											IF arrAxisCtrl[AxiseNo.AxisName.TailCurlRetracting].Cmd.arrbRealPoint[1] THEN
												arrAxisCtrl[AxiseNo.AxisName.TailCurlRetracting].Cmd.iGoSetPos:=0;
												//TailCurlRetMark:=FALSE;//尾卷夹电芯伸缩力矩判断标志
											ELSE
												arrAxisCtrl[AxiseNo.AxisName.TailCurlRetracting].Cmd.iGoSetPos:=1;//尾卷夹电芯伸缩移至初始位
												//TailCurlRetMark:=TRUE;//尾卷夹电芯伸缩力矩判断标志
											END_IF
										END_IF				
										IF 	arrAxisCtrl[AxiseNo.AxisName.TailCurlLine].Status.Homed AND arrAxisCtrl[AxiseNo.AxisName.TailCurlLine].Status.NoMoving THEN
											IF arrAxisCtrl[AxiseNo.AxisName.TailCurlLine].Cmd.arrbRealPoint[3] THEN
												TailCurlTorMark:=FALSE;//尾卷夹电芯平移力矩判断标志位
												bFlgGMEndIng:=FALSE;//拉膜中
												arrAxisCtrl[AxiseNo.AxisName.TailCurlLine].Cmd.iGoSetPos:=0;
											ELSE
												arrAxisCtrl[AxiseNo.AxisName.TailCurlLine].Cmd.iGoSetPos:=3;//尾卷夹电芯平移至拉膜位
												bFlgGMEndIng:=TRUE;//拉膜中
												TailCurlTorMark:=TRUE;//尾卷夹电芯平移力矩判断标志位
											END_IF
										END_IF	
										
				(*					
							//验证：夹膜位更改			
										
										IF 	arrAxis[AxiseNo.AxisName.TailCurlSEPTALine].Status.Homed AND arrAxis[AxiseNo.AxisName.TailCurlSEPTALine].Status.NotMoving THEN
											IF arrAxisCtrl[AxiseNo.AxisName.TailCurlSEPTALine].Cmd.arrbRealPoint[4] THEN
												arrAxisCtrl[AxiseNo.AxisName.TailCurlSEPTALine].Cmd.iGoSetPos:=0;
												TailCurlSEPTATorMark:=FALSE;//夹膜平移力矩判断标志
											ELSE
												arrAxisCtrl[AxiseNo.AxisName.TailCurlSEPTALine].Cmd.iGoSetPos:=4;//尾卷夹膜平移至夹膜
												
												TailCurlSEPTATorMark:=TRUE;//夹膜平移力矩判断标志
											END_IF
										END_IF		
		*)
									
										
										
										IF arrAxisCtrl[AxiseNo.AxisName.TailCurlLine].Status.fSetPos<=  arrAxisPar[AxiseNo.AxisName.TailCurlLine].arrTargetPoint[8] THEN
													IF arrAxis[AxiseNo.AxisName.TailCurlWhirling].Status.Homed AND arrAxisCtrl[AxiseNo.AxisName.TailCurlWhirling].Status.NoMoving THEN
																IF arrAxisCtrl[AxiseNo.AxisName.TailCurlWhirling].Cmd.arrbRealPoint[3] THEN
																	arrAxisCtrl[AxiseNo.AxisName.TailCurlWhirling].Cmd.iGoSetPos:=0;
																ELSE
																	arrAxisCtrl[AxiseNo.AxisName.TailCurlWhirling].Cmd.iGoSetPos:=3;
																END_IF						
												END_IF											
										END_IF
										
								END_IF																	
								IF 	(* arrAxisCtrl[AxiseNo.AxisName.TailCurlSEPTALine].Cmd.arrbRealPoint[4] AND*) arrAxisCtrl[AxiseNo.AxisName.TailCurlRetracting].Cmd.arrbRealPoint[1] AND arrAxisCtrl[AxiseNo.AxisName.TailCurlLine].Cmd.arrbRealPoint[3] AND arrAxisCtrl[AxiseNo.AxisName.TailCurlWhirling].Cmd.arrbRealPoint[3] THEN
											tailCult_GearInMultiMaster.Enable:=FALSE;//启动尾卷拉膜凸轮耦合
											IF Mach_Control.WJ_b.SinStepMode THEN//尾卷单步模式
												TailCurlSinStep:=TRUE;
											ELSE
												TailCurlSinStep:=FALSE;
											END_IF
											fbGearInGMvirbEnable:=FALSE;
											arrAxisCtrl[AxiseNo.AxisName.TailCurlLine].Cmd.fOverride:=100;									
											TailCurlStep3:=160;
											LMcount:=LMcount+1;
								END_IF	
						END_IF
		
				151:	
								
								IF NOT TailCurlSinStep THEN			
										IF arrAxis[AxiseNo.AxisName.TailCurlWhirling].Status.Homed AND arrAxisCtrl[AxiseNo.AxisName.TailCurlWhirling].Status.NoMoving THEN
													IF arrAxisCtrl[AxiseNo.AxisName.TailCurlWhirling].Cmd.arrbRealPoint[3] THEN
														arrAxisCtrl[AxiseNo.AxisName.TailCurlWhirling].Cmd.iGoSetPos:=0;
														IF Mach_Control.WJ_b.SinStepMode THEN//尾卷单步模式
															TailCurlSinStep:=TRUE;
														ELSE
															TailCurlSinStep:=FALSE;
														END_IF	
														TailCurlStep3:=160;
													ELSE
														arrAxisCtrl[AxiseNo.AxisName.TailCurlWhirling].Cmd.iGoSetPos:=3;
													END_IF						
									END_IF
								END_IF
				160://左、右压刀开合至张开位
					IF NOT TailCurlSinStep THEN		
								arrAxisCtrl[AxiseNo.AxisName.TailCurlLine].Cmd.fOverride:=100;
								//Par.stDT_date.iTargetTorqueBLXS:=3;		
								IF 	arrAxisCtrl[AxiseNo.AxisName.LeftYDUpDown].Status.Homed AND arrAxisCtrl[AxiseNo.AxisName.LeftYDUpDown].Status.NoMoving THEN
									IF arrAxisCtrl[AxiseNo.AxisName.LeftYDUpDown].Cmd.arrbRealPoint[2] THEN
										arrAxisCtrl[AxiseNo.AxisName.LeftYDUpDown].Cmd.iGoSetPos:=0;
									ELSE
										arrAxisCtrl[AxiseNo.AxisName.LeftYDUpDown].Cmd.iGoSetPos:=2;//左压刀升降轴上升至下料高度
									END_IF
								END_IF					
								IF 	arrAxisCtrl[AxiseNo.AxisName.RightYDUpDown].Status.Homed AND arrAxisCtrl[AxiseNo.AxisName.RightYDUpDown].Status.NoMoving THEN
									IF arrAxisCtrl[AxiseNo.AxisName.RightYDUpDown].Cmd.arrbRealPoint[2] THEN
										arrAxisCtrl[AxiseNo.AxisName.RightYDUpDown].Cmd.iGoSetPos:=0;
									ELSE
										arrAxisCtrl[AxiseNo.AxisName.RightYDUpDown].Cmd.iGoSetPos:=2;//右压好升降上升至下料高度
									END_IF
								END_IF		
								
								IF 	arrAxisCtrl[AxiseNo.AxisName.TailCurlSEPTAUpDown].Status.Homed AND arrAxisCtrl[AxiseNo.AxisName.TailCurlSEPTAUpDown].Status.NoMoving THEN
									IF arrAxisCtrl[AxiseNo.AxisName.TailCurlSEPTAUpDown].Cmd.arrbRealPoint[2] THEN
										arrAxisCtrl[AxiseNo.AxisName.TailCurlSEPTAUpDown].Cmd.iGoSetPos:=0;
									ELSE
										arrAxisCtrl[AxiseNo.AxisName.TailCurlSEPTAUpDown].Cmd.iGoSetPos:=2;//
									END_IF
								END_IF					
								IF 	arrAxisCtrl[AxiseNo.AxisName.TailCurlUpDown].Status.Homed AND arrAxisCtrl[AxiseNo.AxisName.TailCurlUpDown].Status.NoMoving THEN
									IF arrAxisCtrl[AxiseNo.AxisName.TailCurlUpDown].Cmd.arrbRealPoint[2] THEN
										arrAxisCtrl[AxiseNo.AxisName.TailCurlUpDown].Cmd.iGoSetPos:=0;
									ELSE
										arrAxisCtrl[AxiseNo.AxisName.TailCurlUpDown].Cmd.iGoSetPos:=2;//
									END_IF
								END_IF			
								
								
								IF arrAxisCtrl[AxiseNo.AxisName.TailCurlSEPTAUpDown].Cmd.arrbRealPoint[2]  AND arrAxisCtrl[AxiseNo.AxisName.TailCurlUpDown].Cmd.arrbRealPoint[2] AND
									arrAxisCtrl[AxiseNo.AxisName.LeftYDUpDown].Cmd.arrbRealPoint[2] AND arrAxisCtrl[AxiseNo.AxisName.RightYDUpDown].Cmd.arrbRealPoint[2]  THEN
									IF Mach_Control.WJ_b.SinStepMode THEN//尾卷单步模式
										TailCurlSinStep:=TRUE;
									ELSE
										TailCurlSinStep:=FALSE;
									END_IF		
									TailCurlStep3:=170;
								END_IF
						END_IF		
	
				170:
						IF NOT TailCurlSinStep THEN	
							arrCyCtrl[arrCyNo.ElectValveName.PoleSplintVacuum_D].Cmd.bON:=TRUE;//夹膜下夹板真空	
							arrCyCtrl[arrCyNo.CylinderName.PoleSplintCy_D].Cmd.bON:=TRUE;//夹膜下夹板上升
								IF arrCyCtrl[arrCyNo.CylinderName.PoleSplintCy_D].Status.ONState THEN
									IF Mach_Control.WJ_b.SinStepMode THEN//尾卷单步模式
										TailCurlSinStep:=TRUE;
									ELSE
										TailCurlSinStep:=FALSE;
									END_IF									
									TailCurlStep3:=180;	
								END_IF	
						END_IF		
							
			180:
					
						IF NOT TailCurlSinStep THEN	
							arrCyCtrl[arrCyNo.CylinderName.PreDiaph].Cmd.bON:=TRUE;//叠台压隔膜气缸
							IF arrCyCtrl[arrCyNo.CylinderName.PreDiaph].Status.ONState THEN
										IF Mach_Control.WJ_b.SinStepMode THEN//尾卷单步模式
											TailCurlSinStep:=TRUE;
										ELSE
											TailCurlSinStep:=FALSE;
										END_IF							
										TailCurlStep3:=181;	
							END_IF	
						END_IF	
			181:						
						IF NOT TailCurlSinStep THEN	
									IF 	arrAxisCtrl[AxiseNo.AxisName.DTUpDown].Status.Homed AND arrAxisCtrl[AxiseNo.AxisName.DTUpDown].Status.NoMoving THEN
										IF arrAxisCtrl[AxiseNo.AxisName.DTUpDown].Cmd.arrbRealPoint[1] THEN
											arrAxisCtrl[AxiseNo.AxisName.DTUpDown].Cmd.iGoSetPos:=0;
												IF Mach_Control.DT_b.DT_Chesoe THEN
													DT_Readydown:=TRUE;	
												ELSE
													DT_Readydown:=FALSE;	
												END_IF
	
												IF Mach_Control.WJ_b.SinStepMode THEN//尾卷单步模式
													TailCurlSinStep:=TRUE;
												ELSE
													TailCurlSinStep:=FALSE;
												END_IF													
																								
												TailCurlStep3:=182;	
										ELSE
											arrAxisCtrl[AxiseNo.AxisName.DTUpDown].Cmd.iGoSetPos:=1;//叠台升降上升至初始位
									END_IF
							END_IF
					END_IF
			182:
						IF NOT DT_Readydown THEN
							TailCurlStep3:=185;
						END_IF
			185://左、右压刀开合移至初始位，叠台上升至初始位
						IF NOT TailCurlSinStep THEN		
									IF 	arrAxisCtrl[AxiseNo.AxisName.LeftYDLine].Status.Homed AND arrAxisCtrl[AxiseNo.AxisName.LeftYDLine].Status.NoMoving THEN
										IF arrAxisCtrl[AxiseNo.AxisName.LeftYDLine].Cmd.arrbRealPoint[1] THEN
											arrAxisCtrl[AxiseNo.AxisName.LeftYDLine].Cmd.iGoSetPos:=0;
										ELSE
											arrAxisCtrl[AxiseNo.AxisName.LeftYDLine].Cmd.iGoSetPos:=1;//左压刀开合至初始位
										END_IF
									END_IF					
									IF 	arrAxisCtrl[AxiseNo.AxisName.RightYDLine].Status.Homed AND arrAxisCtrl[AxiseNo.AxisName.RightYDLine].Status.NoMoving THEN
										IF arrAxisCtrl[AxiseNo.AxisName.RightYDLine].Cmd.arrbRealPoint[1] THEN
											arrAxisCtrl[AxiseNo.AxisName.RightYDLine].Cmd.iGoSetPos:=0;
										ELSE
											arrAxisCtrl[AxiseNo.AxisName.RightYDLine].Cmd.iGoSetPos:=1;//右压刀开合至初始位
										END_IF
									END_IF
									IF 	arrAxisCtrl[AxiseNo.AxisName.DTUpDown].Status.Homed AND arrAxisCtrl[AxiseNo.AxisName.DTUpDown].Status.NoMoving THEN
										IF arrAxisCtrl[AxiseNo.AxisName.DTUpDown].Cmd.arrbRealPoint[1] THEN
											arrAxisCtrl[AxiseNo.AxisName.DTUpDown].Cmd.iGoSetPos:=0;
										ELSE
											arrAxisCtrl[AxiseNo.AxisName.DTUpDown].Cmd.iGoSetPos:=1;//叠台升降上升至初始位
										END_IF
									END_IF
									IF 	arrAxisCtrl[AxiseNo.AxisName.LeftYDLine].Cmd.arrbRealPoint[1] AND arrAxisCtrl[AxiseNo.AxisName.RightYDLine].Cmd.arrbRealPoint[1] AND 
										arrAxisCtrl[AxiseNo.AxisName.DTUpDown].Cmd.arrbRealPoint[1] THEN
												TailCurlStep3:=190;
												IF Mach_Control.WJ_b.SinStepMode THEN//尾卷单步模式
													TailCurlSinStep:=TRUE;
												ELSE
													TailCurlSinStep:=FALSE;
												END_IF	
									END_IF	
						END_IF
				
					



				190://左、右压刀升降下降至初始位，压隔膜
						IF NOT TailCurlSinStep THEN			
									IF 	arrAxisCtrl[AxiseNo.AxisName.LeftYDUpDown].Status.Homed AND arrAxisCtrl[AxiseNo.AxisName.LeftYDUpDown].Status.NoMoving THEN
										IF arrAxisCtrl[AxiseNo.AxisName.LeftYDUpDown].Cmd.arrbRealPoint[1] THEN
											arrAxisCtrl[AxiseNo.AxisName.LeftYDUpDown].Cmd.iGoSetPos:=0;
										ELSE
											arrAxisCtrl[AxiseNo.AxisName.LeftYDUpDown].Cmd.iGoSetPos:=1;//左压刀升降轴下降至初始高度
										END_IF
									END_IF					
									IF 	arrAxisCtrl[AxiseNo.AxisName.RightYDUpDown].Status.Homed AND arrAxisCtrl[AxiseNo.AxisName.RightYDUpDown].Status.NoMoving THEN
										IF arrAxisCtrl[AxiseNo.AxisName.RightYDUpDown].Cmd.arrbRealPoint[1] THEN
											arrAxisCtrl[AxiseNo.AxisName.RightYDUpDown].Cmd.iGoSetPos:=0;
										ELSE
											arrAxisCtrl[AxiseNo.AxisName.RightYDUpDown].Cmd.iGoSetPos:=1;//右压好升降下降至初始高度
										END_IF
									END_IF				
									IF arrAxisCtrl[AxiseNo.AxisName.LeftYDUpDown].Cmd.arrbRealPoint[1] AND arrAxisCtrl[AxiseNo.AxisName.RightYDUpDown].Cmd.arrbRealPoint[1] THEN
										IF Mach_Control.WJ_b.SinStepMode THEN//尾卷单步模式
											TailCurlSinStep:=TRUE;
										ELSE
											TailCurlSinStep:=FALSE;
										END_IF											
										TailCurlStep3:=200;
										hot_time_ton.IN:=FALSE;
									END_IF
						END_IF
						
					(*200:
						Mach_Control.WJ_b.HotCut:=TRUE;//启动热切
						WJ_TON[1].IN:=TRUE;
						TailCurlStep3:=201;		
					
						
				201://热切丝加热、热切升降气缸下降，切隔膜///////////////////////////////
					IF NOT TailCurlSinStep THEN	
					arrCyCtrl[arrCyNo.CylinderName.PoleHotCutterCy].Cmd.bON:=TRUE;//隔膜热切升降气缸伸出
								IF arrCyCtrl[arrCyNo.CylinderName.PoleHotCutterCy].Status.ONState  THEN
										Mach_Control.WJ_b.HotCut:=FALSE;//启动热切
						                WJ_TON[1].IN:=FALSE;
							IF Mach_Control.WJ_b.SinStepMode THEN//尾卷单步模式
								TailCurlSinStep:=TRUE;
							ELSE
								TailCurlSinStep:=FALSE;
							END_IF							
									TailCurlStep3:=205;	
								END_IF	
					END_IF	*)
				
				
			
					
				
				
				
				
				
				205://热切升降气缸下降/////////////////////////////////////////
					IF NOT TailCurlSinStep THEN	
						arrCyCtrl[arrCyNo.CylinderName.PoleHotCutterCy].Cmd.bOFF:=TRUE;//隔膜热切升降气缸缩回	
							IF arrCyCtrl[arrCyNo.CylinderName.PoleHotCutterCy].Status.OFFState THEN
								IF Mach_Control.WJ_b.SinStepMode THEN//尾卷单步模式
									TailCurlSinStep:=TRUE;
								ELSE
									TailCurlSinStep:=FALSE;
								END_IF									
								TailCurlStep3:=206;	
							END_IF	
					END_IF		
				206://叠台真空打开
					arrCyCtrl[arrCyNo.ElectValveName.DTVacuum].Cmd.bON:=TRUE;
					arrCyCtrl[arrCyNo.ElectValveName.DTVacuum].Cmd.bOFF:=FALSE;
					TailCurlStep3:=207;	
				207:
					CellMemory[Mach_Control.WJ_b.WJ_Memory]:=CellMemory[Mach_Control.DT_b.DT_Memory];
					MEMSET(ADR(CellMemory[Mach_Control.DT_b.DT_Memory]),0,SIZEOF(CellMemory[Mach_Control.DT_b.DT_Memory]));
					TailCurlStep3:=210;
		
				210:
					
						IF NOT TailCurlSinStep THEN	
							arrCyCtrl[arrCyNo.CylinderName.PreDiaph].Cmd.bOFF:=TRUE;//
							IF arrCyCtrl[arrCyNo.CylinderName.PreDiaph].Status.OFFState THEN
								IF Mach_Control.WJ_b.SinStepMode THEN//尾卷单步模式
									TailCurlSinStep:=TRUE;
								ELSE
									TailCurlSinStep:=FALSE;
								END_IF									
								TailCurlStep3:=211;	
							END_IF	
						END_IF	
				211:
					IF 	arrAxisCtrl[AxiseNo.AxisName.TailCurlUpDown].Status.Homed AND arrAxisCtrl[AxiseNo.AxisName.TailCurlUpDown].Status.NoMoving THEN
						IF arrAxisCtrl[AxiseNo.AxisName.TailCurlUpDown].Cmd.arrbRealPoint[5] THEN
							arrAxisCtrl[AxiseNo.AxisName.TailCurlUpDown].Cmd.iGoSetPos:=0;
							TailCurlStep3:=213;	
						ELSE
							arrAxisCtrl[AxiseNo.AxisName.TailCurlUpDown].Cmd.iGoSetPos:=5;//尾卷夹膜升降轴尾卷高度
						END_IF
					END_IF		
				

				213:
						IF NOT TailCurlSinStep THEN				
						IF 	arrAxisCtrl[AxiseNo.AxisName.TailCurlLine].Status.Homed AND arrAxisCtrl[AxiseNo.AxisName.TailCurlLine].Status.NoMoving THEN
							IF arrAxisCtrl[AxiseNo.AxisName.TailCurlLine].Cmd.arrbRealPoint[7] THEN
								arrAxisCtrl[AxiseNo.AxisName.TailCurlLine].Cmd.iGoSetPos:=0;
								IF Mach_Control.WJ_b.SinStepMode THEN//尾卷单步模式
									TailCurlSinStep:=TRUE;
								ELSE
									TailCurlSinStep:=FALSE;
								END_IF									
								TailCurlStep3:=215;
							ELSE
								arrAxisCtrl[AxiseNo.AxisName.TailCurlLine].Cmd.iGoSetPos:=7;//尾卷夹电芯平移至回拉膜位
							END_IF
						END_IF	
						END_IF
  
			
						
						
                215://尾卷夹电芯平移至上尾卷电芯位，同时开始耦合
						IF NOT TailCurlSinStep THEN			
								tailCurlGearInEnable:=TRUE;//电子齿轮耦合
								IF 	tailCurl_GearIn.InGear AND arrAxisCtrl[AxiseNo.AxisName.TailCurlLine].Status.Homed AND arrAxisCtrl[AxiseNo.AxisName.TailCurlLine].Status.NoMoving AND
                                        arrAxisCtrl[AxiseNo.AxisName.LCurlingneedleLine].Cmd.arrbRealPoint[1]  AND arrAxisCtrl[AxiseNo.AxisName.SCurlingneedleLine].Cmd.arrbRealPoint[1] AND
                                       arrAxisCtrl[AxiseNo.AxisName.TailCurlWhirling].Cmd.arrbRealPoint[1]   THEN
									IF arrAxisCtrl[AxiseNo.AxisName.TailCurlLine].Cmd.arrbRealPoint[4] THEN
										arrAxisCtrl[AxiseNo.AxisName.TailCurlLine].Cmd.iGoSetPos:=0;
										tailCurlGearInEnable:=FALSE;//电子齿轮耦合
										IF Mach_Control.WJ_b.SinStepMode THEN//尾卷单步模式
											TailCurlSinStep:=TRUE;
										ELSE
											TailCurlSinStep:=FALSE;
										END_IF												
										TailCurlStep3:=217;
										TailCurlStep6:=10;//启动判断夹膜平移是否已经在安全位置叠台下料完成	
										WJ_TON[6].IN:=FALSE;
									ELSE
										arrAxisCtrl[AxiseNo.AxisName.TailCurlLine].Cmd.iGoSetPos:=4;//尾卷夹电芯平移至上尾卷电芯位
									END_IF
								END_IF		
						END_IF	
               
				217:	
					 WJ_TON[6].IN:=TRUE;
					Mach_Control.WJ_b.TailCurlSEPTALineSavePos[1]:=arrAxis[AxiseNo.AxisName.TailCurlSEPTALine].NcToPlc.ActPos;
					arrAxisCtrl[AxiseNo.AxisName.TailCurlSEPTALine].Cmd.bMoveRel:=FALSE;
					IF WJ_TON[6].Q THEN
						TailCurlStep3:=218;
						 WJ_TON[6].IN:=FALSE;
					 END_IF	
				 
				218:
				IF NOT TailCurlSinStep THEN	
				IF Mach_Control.WJ_b.TailCurlSEPTALineSavePos[1] -arrAxis[AxiseNo.AxisName.TailCurlSEPTALine].NcToPlc.ActPos>=4.9 
					AND arrAxisCtrl[AxiseNo.AxisName.TailCurlSEPTALine].Status.NoMoving THEN
						IF Mach_Control.WJ_b.SinStepMode THEN//尾卷单步模式
								TailCurlSinStep:=TRUE;
						ELSE
								TailCurlSinStep:=FALSE;
						END_IF
					TailCurlStep3:=220;
				ELSIF NOT (Mach_Control.WJ_b.TailCurlSEPTALineSavePos[1] -arrAxis[AxiseNo.AxisName.TailCurlSEPTALine].NcToPlc.ActPos >=4.9 )
						AND arrAxisCtrl[AxiseNo.AxisName.TailCurlSEPTALine].Status.NoMoving THEN
						IF NOT arrAxisCtrl[AxiseNo.AxisName.TailCurlSEPTALine].Status.Error 
							AND arrAxis[AxiseNo.AxisName.TailCurlSEPTALine].Status.Homed 
							AND arrAxisCtrl[AxiseNo.AxisName.TailCurlSEPTALine].Status.Enabled 
							AND arrAxisCtrl[AxiseNo.AxisName.TailCurlSEPTALine].Status.NoMoving THEN
								arrAxisPar[AxiseNo.AxisName.TailCurlSEPTALine].fVelocity_of_Rel:=20;
								arrAxisCtrl[AxiseNo.AxisName.TailCurlSEPTALine].Cmd.fPosition_of_Rel:=-5;
								arrAxisCtrl[AxiseNo.AxisName.TailCurlSEPTALine].Cmd.bMoveRel:=TRUE;
						END_IF
				END_IF
				END_IF
						
						
						
				220://长、短卷针旋转到初始位，长、短卷针气缸张开/////////
						IF NOT TailCurlSinStep THEN		
								arrCyCtrl[arrCyNo.ElectValveName.WJ_blow		].Cmd.bON:=	TRUE	;//	夹膜电芯吹气	
						
								arrCyCtrl[arrCyNo.CylinderName.CurlingSplintCy_L].Cmd.bOFF:=TRUE;//尾卷长卷针张开
								arrCyCtrl[arrCyNo.CylinderName.CurlingSplintCy_S].Cmd.bOFF:=TRUE;//尾卷短卷针张开
								arrCyCtrl[arrCyNo.ElectValveName.WJShortvacuum].Cmd.bON:=TRUE;//短卷针张开真空开
								IF 	arrAxisCtrl[AxiseNo.AxisName.LCurlingneedleWhirling].Status.Homed AND arrAxisCtrl[AxiseNo.AxisName.LCurlingneedleWhirling].Status.NoMoving THEN
									IF arrAxisCtrl[AxiseNo.AxisName.LCurlingneedleWhirling].Cmd.arrbRealPoint[1] THEN
										arrAxisCtrl[AxiseNo.AxisName.LCurlingneedleWhirling].Cmd.iGoSetPos:=0;
									ELSE
										arrAxisCtrl[AxiseNo.AxisName.LCurlingneedleWhirling].Cmd.iGoSetPos:=1;//长卷针旋转至初始位
									END_IF
								END_IF										
								IF 	arrAxisCtrl[AxiseNo.AxisName.SCurlingneedleWhirling].Status.Homed AND arrAxisCtrl[AxiseNo.AxisName.SCurlingneedleWhirling].Status.NoMoving THEN
									IF arrAxisCtrl[AxiseNo.AxisName.SCurlingneedleWhirling].Cmd.arrbRealPoint[1] THEN
										arrAxisCtrl[AxiseNo.AxisName.SCurlingneedleWhirling].Cmd.iGoSetPos:=0;
									ELSE
										arrAxisCtrl[AxiseNo.AxisName.SCurlingneedleWhirling].Cmd.iGoSetPos:=1;//短卷针旋转至初始位
									END_IF
								END_IF
								
								
								IF 	arrAxisCtrl[AxiseNo.AxisName.TailCurlUpDown].Status.Homed AND arrAxisCtrl[AxiseNo.AxisName.TailCurlUpDown].Status.NoMoving THEN
									IF arrAxisCtrl[AxiseNo.AxisName.TailCurlUpDown].Cmd.arrbRealPoint[5] THEN
										arrAxisCtrl[AxiseNo.AxisName.TailCurlUpDown].Cmd.iGoSetPos:=0;
									ELSE
										arrAxisCtrl[AxiseNo.AxisName.TailCurlUpDown].Cmd.iGoSetPos:=5;//尾卷夹膜升降轴尾卷高度
									END_IF
								END_IF	
								
								
								
								IF 	arrAxisCtrl[AxiseNo.AxisName.LCurlingneedleWhirling].Cmd.arrbRealPoint[1] AND 	arrAxisCtrl[AxiseNo.AxisName.SCurlingneedleWhirling].Cmd.arrbRealPoint[1] AND
									arrAxisCtrl[AxiseNo.AxisName.TailCurlUpDown].Cmd.arrbRealPoint[5]  AND 
                                    					arrCyCtrl[arrCyNo.CylinderName.CurlingSplintCy_L].Status.OFFState AND arrCyCtrl[arrCyNo.CylinderName.CurlingSplintCy_S].Status.OFFState THEN
										IF Mach_Control.WJ_b.SinStepMode THEN//尾卷单步模式
											TailCurlSinStep:=TRUE;
										ELSE
											TailCurlSinStep:=FALSE;
										END_IF	
									CurlingneedleLineEnable:=FALSE;//长、短卷针平移电子齿轮耦合启动																
									TailCurlStep3:=223;
								END_IF	
						END_IF	
                






			223://长卷针去夹电芯位
				IF NOT TailCurlSinStep THEN		
								
								IF 	arrAxisCtrl[AxiseNo.AxisName.LCurlingneedleLine].Status.Homed  
								AND arrAxisCtrl[AxiseNo.AxisName.LCurlingneedleWhirling].Cmd.arrbRealPoint[1]
								AND arrCyCtrl[arrCyNo.CylinderName.CurlingSplintCy_L].Status.OFFState
                                AND  arrAxisCtrl[AxiseNo.AxisName.LCurlingneedleWhirling].Io.biHomeSwitch  THEN
											IF arrAxisCtrl[AxiseNo.AxisName.LCurlingneedleLine].Cmd.arrbRealPoint[2] AND arrAxisCtrl[AxiseNo.AxisName.LCurlingneedleLine].Status.NoMoving  THEN
												arrAxisCtrl[AxiseNo.AxisName.LCurlingneedleLine].Cmd.iGoSetPos:=0;
											ELSE
												arrAxisCtrl[AxiseNo.AxisName.LCurlingneedleLine].Cmd.iGoSetPos:=2;
											END_IF
								ELSE
										Mach_Control.WJ_b.Error[9]:=TRUE;	//长卷针去夹电芯位时条件不满足报警													
								END_IF
										
								IF 	arrAxisCtrl[AxiseNo.AxisName.LCurlingneedleLine].Cmd.arrbRealPoint[2] AND arrAxisCtrl[AxiseNo.AxisName.LCurlingneedleWhirling].Cmd.arrbRealPoint[1]  THEN
										IF Mach_Control.WJ_b.SinStepMode THEN//尾卷单步模式
											TailCurlSinStep:=TRUE;
										ELSE
											TailCurlSinStep:=FALSE;
										END_IF																	
									TailCurlStep3:=225;
									TON_TailCurl[2].IN:=FALSE;
								END_IF	
						END_IF			
			225:
			
			
						IF NOT TailCurlSinStep THEN	
								 
													IF NOT TON_TailCurl[2].Q THEN					
																arrCyCtrl[arrCyNo.CylinderName.CurlingSplintCy_L].Cmd.bON:=TRUE;//尾卷长卷针夹紧	
																TON_TailCurl[2].IN:=TRUE;			
													ELSE
														TON_TailCurl[2].IN:=FALSE;
														IF Mach_Control.WJ_b.SinStepMode THEN//尾卷单步模式
															TailCurlSinStep:=TRUE;
														ELSE
															TailCurlSinStep:=FALSE;
														END_IF							
														TailCurlStep3:=227;	
												END_IF
									
						END_IF

			227://短卷针去夹电芯位
	
						
					IF NOT TailCurlSinStep THEN													
								IF 	arrAxisCtrl[AxiseNo.AxisName.SCurlingneedleLine].Status.Homed  
									AND arrAxisCtrl[AxiseNo.AxisName.SCurlingneedleWhirling].Cmd.arrbRealPoint[1] AND  arrCyCtrl[arrCyNo.CylinderName.CurlingSplintCy_S].Status.OFFState 
									AND  arrCyCtrl[arrCyNo.ElectValveName.WJShortvacuum].Io.DOStatus1
                                    AND  arrAxisCtrl[AxiseNo.AxisName.SCurlingneedleWhirling].Io.biHomeSwitch THEN
												IF arrAxisCtrl[AxiseNo.AxisName.SCurlingneedleLine].Cmd.arrbRealPoint[2] AND arrAxisCtrl[AxiseNo.AxisName.SCurlingneedleLine].Status.NoMoving  THEN
													arrAxisCtrl[AxiseNo.AxisName.SCurlingneedleLine].Cmd.iGoSetPos:=0;
												ELSE
													arrAxisCtrl[AxiseNo.AxisName.SCurlingneedleLine].Cmd.iGoSetPos:=2;
												END_IF
								ELSE
										Mach_Control.WJ_b.Error[10]:=TRUE;	//短卷针去夹电芯位时条件不满足报警										
												
								END_IF

								IF 		arrAxisCtrl[AxiseNo.AxisName.SCurlingneedleLine].Cmd.arrbRealPoint[2] AND arrAxisCtrl[AxiseNo.AxisName.SCurlingneedleWhirling].Cmd.arrbRealPoint[1] THEN
										IF Mach_Control.WJ_b.SinStepMode THEN//尾卷单步模式
											TailCurlSinStep:=TRUE;
										ELSE
											TailCurlSinStep:=FALSE;
										END_IF																	
									TailCurlStep3:=230;
									TON_TailCurl[4].IN:=FALSE;
								END_IF	
						END_IF		
						
			
						
				230://短卷针夹爪气缸夹紧
						IF NOT TailCurlSinStep THEN	
							     
													IF NOT TON_TailCurl[4].Q THEN
														arrCyCtrl[arrCyNo.ElectValveName.WJShortvacuum].Cmd.bOFF:=TRUE;//短卷针张开真空关
														arrCyCtrl[arrCyNo.CylinderName.CurlingSplintCy_S].Cmd.bON:=TRUE;//尾卷短卷针夹紧	
														
														TON_TailCurl[4].IN:=TRUE;							
													ELSE
														TON_TailCurl[4].IN:=FALSE;
														IF Mach_Control.WJ_b.SinStepMode THEN//尾卷单步模式
															TailCurlSinStep:=TRUE;
														ELSE
															TailCurlSinStep:=FALSE;
														END_IF							
														TailCurlStep3:=235;	
														TON_TailCurl[6].IN:=FALSE;
												END_IF
										
						END_IF
				               
				235:
				Mach_Control.WJ_b.TailCurlSEPTALineSavePos[2]:=arrAxis[AxiseNo.AxisName.TailCurlSEPTALine].NcToPlc.ActPos;
				TailCurlStep3:=238;

				238:
				IF NOT TailCurlSinStep THEN	
				IF arrAxis[AxiseNo.AxisName.TailCurlSEPTALine].NcToPlc.ActPos-Mach_Control.WJ_b.TailCurlSEPTALineSavePos[2] >=4.9 
					AND arrAxisCtrl[AxiseNo.AxisName.TailCurlSEPTALine].Status.NoMoving THEN
						IF Mach_Control.WJ_b.SinStepMode THEN//尾卷单步模式
								TailCurlSinStep:=TRUE;
						ELSE
								TailCurlSinStep:=FALSE;
						END_IF
					TailCurlStep3:=240;
				ELSIF NOT (arrAxis[AxiseNo.AxisName.TailCurlSEPTALine].NcToPlc.ActPos-Mach_Control.WJ_b.TailCurlSEPTALineSavePos[2] >=4.9 )
					AND arrAxisCtrl[AxiseNo.AxisName.TailCurlSEPTALine].Status.NoMoving THEN
						IF NOT arrAxisCtrl[AxiseNo.AxisName.TailCurlSEPTALine].Status.Error 
							AND arrAxis[AxiseNo.AxisName.TailCurlSEPTALine].Status.Homed 
							AND arrAxisCtrl[AxiseNo.AxisName.TailCurlSEPTALine].Status.Enabled 
							AND arrAxisCtrl[AxiseNo.AxisName.TailCurlSEPTALine].Status.NoMoving THEN
								arrAxisPar[AxiseNo.AxisName.TailCurlSEPTALine].fVelocity_of_Rel:=20;
								arrAxisCtrl[AxiseNo.AxisName.TailCurlSEPTALine].Cmd.fPosition_of_Rel:=5;
								arrAxisCtrl[AxiseNo.AxisName.TailCurlSEPTALine].Cmd.bMoveRel:=TRUE;
						END_IF
				END_IF
				END_IF
				
				240://尾卷夹电芯气缸开张
						IF NOT TailCurlSinStep THEN	
							arrCyCtrl[arrCyNo.ElectValveName.WJ_blow].Cmd.bOFF:=TRUE;//	夹膜电芯吹气关
							arrCyCtrl[arrCyNo.CylinderName.TailCurlSplintCy].Cmd.bOFF:=TRUE;//尾卷取料夹爪气缸张开
							TON_TailCurl[6].IN:=TRUE;
							IF arrCyCtrl[arrCyNo.CylinderName.TailCurlSplintCy].Status.OFFState AND TON_TailCurl[6].Q	THEN
								IF Mach_Control.WJ_b.SinStepMode THEN//尾卷单步模式
									TailCurlSinStep:=TRUE;
								ELSE
									TailCurlSinStep:=FALSE;
								END_IF						
								TailCurlStep3:=250;
								TON_TailCurl[6].IN:=FALSE;
							END_IF
						END_IF
				250://尾卷夹电芯平移至初始位，启动尾卷
						IF NOT TailCurlSinStep THEN			
									IF 	arrCyCtrl[arrCyNo.CylinderName.TailCurlSplintCy].Status.OFFState AND  arrAxisCtrl[AxiseNo.AxisName.TailCurlLine].Status.Homed AND arrAxisCtrl[AxiseNo.AxisName.TailCurlLine].Status.NoMoving THEN
											IF arrAxisCtrl[AxiseNo.AxisName.TailCurlLine].Cmd.arrbRealPoint[5] THEN
												TailCurlTorMark:=FALSE;//尾卷夹电芯平移力矩判断标志位
												//TailCurlStart:=TRUE;//启动尾卷
												arrAxisCtrl[AxiseNo.AxisName.TailCurlLine].Cmd.iGoSetPos:=0;
											ELSE
												arrAxisCtrl[AxiseNo.AxisName.TailCurlLine].Cmd.iGoSetPos:=5;//尾卷夹电芯平移至初始位
												TailCurlTorMark:=TRUE;//尾卷夹电芯平移力矩判断标志位
											END_IF
									END_IF	
									
									IF arrCyCtrl[arrCyNo.CylinderName.TailCurlSplintCy].Status.OFFState AND  	arrAxisCtrl[AxiseNo.AxisName.TailCurlRetracting].Status.Homed AND arrAxisCtrl[AxiseNo.AxisName.TailCurlRetracting].Status.NoMoving THEN
											IF arrAxisCtrl[AxiseNo.AxisName.TailCurlRetracting].Cmd.arrbRealPoint[1] THEN
												//TailCurlRetMark:=FALSE;//尾卷夹电芯伸缩力矩判断标志
												arrAxisCtrl[AxiseNo.AxisName.TailCurlRetracting].Cmd.iGoSetPos:=0;
											ELSE
												arrAxisCtrl[AxiseNo.AxisName.TailCurlRetracting].Cmd.iGoSetPos:=1;//尾卷夹电芯伸缩移至初始位
												//TailCurlRetMark:=TRUE;//尾卷夹电芯伸缩力矩判断标志
											END_IF
									END_IF		
									
									IF 		arrAxisCtrl[AxiseNo.AxisName.TailCurlLine].Cmd.arrbRealPoint[5] AND arrAxisCtrl[AxiseNo.AxisName.TailCurlLine].Status.NoMoving AND
											 arrAxisCtrl[AxiseNo.AxisName.TailCurlRetracting].Cmd.arrbRealPoint[1] AND  arrAxisCtrl[AxiseNo.AxisName.TailCurlRetracting].Status.NoMoving THEN
													IF Mach_Control.WJ_b.SinStepMode THEN//尾卷单步模式
														TailCurlSinStep:=TRUE;
													ELSE
														TailCurlSinStep:=FALSE;
													END_IF											
													TailCurlStep3:=251;	
													CurlingneedleLineEnable:=TRUE;//长、短卷针平移电子齿轮耦合启动
									END_IF						
						END_IF	
					
						
				251://长、短卷针电子齿轮耦合，移动至尾卷补偿位
						IF NOT TailCurlSinStep THEN		
								
						
								IF 	arrAxisCtrl[AxiseNo.AxisName.LCurlingneedleLine].Status.Homed AND arrAxisCtrl[AxiseNo.AxisName.LCurlingneedleLine].Status.NoMoving AND CurlingneedleLine_GearIn.InGear THEN
									IF arrAxisCtrl[AxiseNo.AxisName.LCurlingneedleLine].Cmd.arrbRealPoint[3] THEN
										arrAxisCtrl[AxiseNo.AxisName.LCurlingneedleLine].Cmd.iGoSetPos:=0;
										CurlingneedleLineEnable:=FALSE;//长、短卷针平移电子齿轮耦合启动
										IF Mach_Control.WJ_b.SinStepMode THEN//尾卷单步模式
											TailCurlSinStep:=TRUE;
										ELSE
											TailCurlSinStep:=FALSE;
										END_IF	
										//IF NOT CurlingneedleLine_GearIn.InGear THEN
											TailCurlStep3:=252;
										//END_IF
									ELSE
										arrAxisCtrl[AxiseNo.AxisName.LCurlingneedleLine].Cmd.iGoSetPos:=3;
									END_IF
								END_IF	
						END_IF
						
		    	252:
					IF NOT CurlingneedleLine_GearIn.InGear AND arrAxisCtrl[AxiseNo.AxisName.SCurlingneedleLine].Status.NoMoving AND 
							(ABS((ABS(arrAxisCtrl[AxiseNo.AxisName.SCurlingneedleLine].Status.fActPos-arrAxisPar[AxiseNo.AxisName.SCurlingneedleLine].arrTargetPoint[2] )-
							ABS(arrAxisPar[AxiseNo.AxisName.LCurlingneedleLine].arrTargetPoint[3]-arrAxisPar[AxiseNo.AxisName.LCurlingneedleLine].arrTargetPoint[2])))<=0.5) THEN
					    TailCurlStep3:=253;
					END_IF
				
				253:
					TailCurlStep0:=50;
					TailCurlStep3:=254;
				254:
					IF TailCurlStep0=6666 THEN
						TailCurlStep3:=255;
					END_IF
				255: 
				  IF  arrAxisCtrl[AxiseNo.AxisName.TailCurlLine].Status.fActPos<=arrAxisPar[AxiseNo.AxisName.TailCurlLine].arrTargetPoint[5]+1 THEN
						TailCurlStart:=TRUE;//启动尾卷
						TailCurlStep3:=256;
				END_IF 	
				256:
					IF NOT TailCurlSinStep THEN	
						IF arrAxis[AxiseNo.AxisName.TailCurlWhirling].Status.Homed AND arrAxisCtrl[AxiseNo.AxisName.TailCurlWhirling].Status.NoMoving THEN
								IF arrAxisCtrl[AxiseNo.AxisName.TailCurlWhirling].Cmd.arrbRealPoint[1] THEN
									arrAxisCtrl[AxiseNo.AxisName.TailCurlWhirling].Cmd.iGoSetPos:=0;
									IF Mach_Control.WJ_b.SinStepMode THEN//尾卷单步模式
										TailCurlSinStep:=TRUE;
									ELSE
										TailCurlSinStep:=FALSE;
									END_IF	
									TailCurlStep3:=260;
								ELSE
									arrAxisCtrl[AxiseNo.AxisName.TailCurlWhirling].Cmd.iGoSetPos:=1;
								END_IF		
						END_IF				
					END_IF					
										
		
				260://等待尾卷完成信号
				
					IF Mach_Control.WJ_b.TailCurlDone (*AND TailCurlStep6=666*) THEN
						TailCurlStart:=FALSE;//启动尾卷
						// Mach_Control.DT_b.OffloadDone:=TRUE;//(已经在TailCurlStep6子程序里置位)
						 arrCyCtrl[arrCyNo.ElectValveName.PoleSplintVacuum_D].Cmd.bOFF:=TRUE;//夹膜下夹板真空	
						IF Mach_Control.WJ_b.SinStepMode THEN//尾卷单步模式
							TailCurlSinStep:=TRUE;
						ELSE
							TailCurlSinStep:=FALSE;
						END_IF
						Mach_Control.WJ_b.TailCurlDone	:=FALSE;						
						TailCurlStep3:=271;
					END_IF
					
				270://尾卷取电芯夹爪气缸平夹紧
						IF NOT TailCurlSinStep THEN				
							arrCyCtrl[arrCyNo.CylinderName.PoleSplintCy_D].Cmd.bOFF:=TRUE;//尾卷取料夹爪气缸夹紧
							IF arrCyCtrl[arrCyNo.CylinderName.PoleSplintCy_D].Status.OFFState THEN
								IF Mach_Control.WJ_b.SinStepMode THEN//尾卷单步模式
									TailCurlSinStep:=TRUE;
								ELSE
									TailCurlSinStep:=FALSE;
								END_IF										
								TailCurlStep3:=271;
							END_IF
						END_IF
				
				271://长、短卷针电子齿轮耦合，移动至尾卷补偿位
						IF NOT TailCurlSinStep THEN		
								CurlingneedleLineEnable:=TRUE;//长、短卷针平移电子齿轮耦合启动
								IF 	arrAxisCtrl[AxiseNo.AxisName.LCurlingneedleLine].Status.Homed AND arrAxisCtrl[AxiseNo.AxisName.LCurlingneedleLine].Status.NoMoving AND CurlingneedleLine_GearIn.InGear  THEN
									IF arrAxisCtrl[AxiseNo.AxisName.LCurlingneedleLine].Cmd.arrbRealPoint[4] THEN
										arrAxisCtrl[AxiseNo.AxisName.LCurlingneedleLine].Cmd.iGoSetPos:=0;
										CurlingneedleLineEnable:=FALSE;//长、短卷针平移电子齿轮耦合启动
										IF Mach_Control.WJ_b.SinStepMode THEN//尾卷单步模式
											TailCurlSinStep:=TRUE;
										ELSE
											TailCurlSinStep:=FALSE;
										END_IF	
										TailCurlStep3:=272;
									ELSE
										arrAxisCtrl[AxiseNo.AxisName.LCurlingneedleLine].Cmd.iGoSetPos:=4;
									END_IF
								END_IF	
						END_IF					
					
				272://尾卷夹电芯升降到尾卷完下电芯位
					IF 	arrAxisCtrl[AxiseNo.AxisName.TailCurlUpDown].Status.Homed AND arrAxisCtrl[AxiseNo.AxisName.TailCurlUpDown].Status.NoMoving THEN
						IF arrAxisCtrl[AxiseNo.AxisName.TailCurlUpDown].Cmd.arrbRealPoint[7] THEN
							arrAxisCtrl[AxiseNo.AxisName.TailCurlUpDown].Cmd.iGoSetPos:=0;
							IF Mach_Control.WJ_b.SinStepMode THEN//尾卷单步模式
								TailCurlSinStep:=TRUE;
							ELSE
								TailCurlSinStep:=FALSE;
							END_IF	
							TailCurlStep3:=275;
						ELSE
							arrAxisCtrl[AxiseNo.AxisName.TailCurlUpDown].Cmd.iGoSetPos:=7;
						END_IF
					END_IF	
	                           
				275://尾卷取电芯夹爪张开，尾卷夹电芯平移至尾卷取电芯位下电芯
					IF NOT TailCurlSinStep THEN		
                               				
							arrCyCtrl[arrCyNo.CylinderName.TailCurlSplintCy].Cmd.bOFF:=TRUE;//尾卷取料夹爪气缸张开
							IF  arrCyCtrl[arrCyNo.CylinderName.TailCurlSplintCy].Status.OFFState AND arrAxisCtrl[AxiseNo.AxisName.TailCurlLine].Status.NoMoving  THEN
								TailCurlStep3:=278;
							END_IF		
						END_IF		
				278:
				     IF NOT TailCurlSinStep THEN	
									IF ABS(arrAxisCtrl[AxiseNo.AxisName.LCurlingneedleWhirling].Status.fActPos - (arrAxisPar[AxiseNo.AxisName.LCurlingneedleWhirling].arrTargetPoint[1]+360)) <=1 AND 					
										arrAxisCtrl[AxiseNo.AxisName.LCurlingneedleWhirling].Status.NoMoving AND arrAxisCtrl[AxiseNo.AxisName.LCurlingneedleWhirling].Io.biHomeSwitch AND
										ABS(arrAxisCtrl[AxiseNo.AxisName.SCurlingneedleWhirling].Status.fActPos - (arrAxisPar[AxiseNo.AxisName.SCurlingneedleWhirling].arrTargetPoint[1]+360))<=1  AND
										arrAxisCtrl[AxiseNo.AxisName.SCurlingneedleWhirling].Status.NoMoving AND arrAxisCtrl[AxiseNo.AxisName.SCurlingneedleWhirling].Io.biHomeSwitch AND
									    arrAxisCtrl[AxiseNo.AxisName.LCurlingneedleWhirling].Io.biHomeSwitch     AND   arrCyCtrl[arrCyNo.CylinderName.TailCurlSplintCy].Status.OFFState AND
                                  		arrCyCtrl[arrCyNo.CylinderName.CurlingSplintCy_L].Status.ONState AND arrCyCtrl[arrCyNo.CylinderName.CurlingSplintCy_S].Status.ONState AND  
                                       NOT  arrCyCtrl[arrCyNo.ElectValveName.WJShortvacuum].Io.DOStatus1  AND 
                                       arrAxisCtrl[AxiseNo.AxisName.TailCurlLine].Status.Homed THEN
																IF arrAxisCtrl[AxiseNo.AxisName.TailCurlLine].Cmd.arrbRealPoint[4] AND arrAxisCtrl[AxiseNo.AxisName.TailCurlLine].Status.NoMoving  THEN
																	arrAxisCtrl[AxiseNo.AxisName.TailCurlLine].Cmd.iGoSetPos:=0;
																		IF Mach_Control.WJ_b.SinStepMode THEN//尾卷单步模式
																			TailCurlSinStep:=TRUE;
																		ELSE
																			TailCurlSinStep:=FALSE;
																		END_IF											
																				TailCurlStep3:=280;
																ELSE
																	arrAxisCtrl[AxiseNo.AxisName.TailCurlLine].Cmd.iGoSetPos:=4;//尾卷夹电芯平移至取电芯位
																END_IF
					
									ELSE
										Mach_Control.WJ_b.Error[7]:=TRUE;//尾卷下料时卷针旋转不满足下料角度----20240116
									END_IF	
				     END_IF	
			(*	279:
					IF arrAxisCtrl[AxiseNo.AxisName.TailCurlLine].Cmd.arrbRealPoint[4] THEN
						arrAxisCtrl[AxiseNo.AxisName.TailCurlLine].Cmd.iGoSetPos:=0;
							IF Mach_Control.WJ_b.SinStepMode THEN//尾卷单步模式
								TailCurlSinStep:=TRUE;
							ELSE
								TailCurlSinStep:=FALSE;
							END_IF											
									TailCurlStep3:=280;
					ELSE
						arrAxisCtrl[AxiseNo.AxisName.TailCurlLine].Cmd.iGoSetPos:=4;//尾卷夹电芯平移至取电芯位
					END_IF*)
				
				280://尾卷取电芯夹爪气缸平夹紧
						IF NOT TailCurlSinStep THEN				
							arrCyCtrl[arrCyNo.CylinderName.TailCurlSplintCy].Cmd.bON:=TRUE;//尾卷取料夹爪气缸夹紧
							IF arrCyCtrl[arrCyNo.CylinderName.TailCurlSplintCy].Io.DIOnSwitch THEN
								arrCyCtrl[arrCyNo.ElectValveName.WJ_blow].Cmd.bON:=TRUE;//	夹膜电芯吹气开
								IF Mach_Control.WJ_b.SinStepMode THEN//尾卷单步模式
									TailCurlSinStep:=TRUE;
								ELSE
									TailCurlSinStep:=FALSE;
								END_IF	
								TailCurlStep3:=283;
							END_IF
						END_IF
				
				283://夹膜打开
						IF NOT TailCurlSinStep THEN				
							arrCyCtrl[arrCyNo.CylinderName.PoleSplintCy_D].Cmd.bOFF:=TRUE;
							
							IF arrCyCtrl[arrCyNo.CylinderName.PoleSplintCy_D].Status.OFFState THEN
								IF Mach_Control.WJ_b.SinStepMode THEN//尾卷单步模式
									TailCurlSinStep:=TRUE;
								ELSE
									TailCurlSinStep:=FALSE;
								END_IF
								//arrCyCtrl[arrCyNo.ElectValveName.WJ_blow].Cmd.bON:=FALSE;//	夹膜电芯吹气关
								//arrCyCtrl[arrCyNo.ElectValveName.WJ_blow].Cmd.bOFF:=TRUE;//	夹膜电芯吹气关										
								TailCurlStep3:=287;
							END_IF
						END_IF
					
				287:	
					IF arrCyCtrl[arrCyNo.CylinderName.PoleSplintCy_D].Status.OFFState AND NOT arrAxisCtrl[AxiseNo.AxisName.TailCurlSEPTALine].Status.Coupled AND 
							NOT arrAxisCtrl[AxiseNo.AxisName.TailCurlSEPTAUpDown].Status.Coupled THEN
						IF 	 arrAxis[AxiseNo.AxisName.TailCurlSEPTALine].Status.Homed AND arrAxisCtrl[AxiseNo.AxisName.TailCurlSEPTALine].Status.NoMoving THEN
							IF arrAxisCtrl[AxiseNo.AxisName.TailCurlSEPTALine].Cmd.arrbRealPoint[1] THEN
								arrAxisCtrl[AxiseNo.AxisName.TailCurlSEPTALine].Cmd.iGoSetPos:=0;
							ELSE
								arrAxisCtrl[AxiseNo.AxisName.TailCurlSEPTALine].Cmd.iGoSetPos:=1;//尾卷夹隔膜平移初始位
							END_IF
						END_IF	
						IF 	 arrAxisCtrl[AxiseNo.AxisName.TailCurlSEPTAUpDown].Status.Homed AND arrAxisCtrl[AxiseNo.AxisName.TailCurlSEPTAUpDown].Status.NoMoving THEN
							IF arrAxisCtrl[AxiseNo.AxisName.TailCurlSEPTAUpDown].Cmd.arrbRealPoint[1] THEN
								arrAxisCtrl[AxiseNo.AxisName.TailCurlSEPTAUpDown].Cmd.iGoSetPos:=0;
							ELSE
								arrAxisCtrl[AxiseNo.AxisName.TailCurlSEPTAUpDown].Cmd.iGoSetPos:=1;//尾卷夹隔膜升降初始位
							END_IF
						END_IF
						IF 	arrAxisCtrl[AxiseNo.AxisName.TailCurlSEPTALine].Cmd.arrbRealPoint[1] AND  arrAxisCtrl[AxiseNo.AxisName.TailCurlSEPTAUpDown].Cmd.arrbRealPoint[1]  THEN
								IF Mach_Control.WJ_b.SinStepMode THEN//尾卷单步模式
									TailCurlSinStep:=TRUE;
								ELSE
									TailCurlSinStep:=FALSE;
								END_IF				
								TailCurlStep3:=290;	
						END_IF	
					END_IF			








					290://尾卷压轮升降气缸收回、平移气缸收回
						IF NOT TailCurlSinStep THEN		
								arrCyCtrl[arrCyNo.CylinderName.TailCurlUpdownCy].Cmd.bOFF:=TRUE;//尾卷压轮升降气缸收回
								IF arrCyCtrl[arrCyNo.CylinderName.TailCurlUpdownCy].Io.DIOFFSwitch THEN
									arrCyCtrl[arrCyNo.CylinderName.TailCurlLineCy].Cmd.bOFF:=TRUE;//尾卷压轮平移气缸收回		
									IF arrCyCtrl[arrCyNo.CylinderName.TailCurlLineCy].Io.DIOFFSwitch THEN
										IF Mach_Control.WJ_b.SinStepMode THEN//尾卷单步模式
											TailCurlSinStep:=TRUE;
										ELSE
											TailCurlSinStep:=FALSE;
										END_IF	
										TailCurlStep3:=300;
									END_IF
								END_IF
						END_IF
				300://长、短卷针夹电芯气缸泄压、长、短卷针伸缩轴移动至初始位
						IF NOT TailCurlSinStep THEN			
									IF NOT TON_TailCurl[3].Q THEN
										arrCyCtrl[arrCyNo.CylinderName.CurlingSplintCy_L].Cmd.bFree:=TRUE;//尾卷长卷针泄压
										arrCyCtrl[arrCyNo.CylinderName.CurlingSplintCy_S].Cmd.bFree:=TRUE;//尾卷短卷针泄压
										//arrCyCtrl[arrCyNo.ElectValveName.WJShortvacuum].Cmd.bON:=TRUE;//短卷针张开真空开
										//arrCyCtrl[arrCyNo.CylinderName.CurlingSplintCy_S_1].Cmd.bOFF:=TRUE;//尾卷短卷针泄压
										TON_TailCurl[3].IN:=TRUE;
									ELSE
										IF 	arrAxisCtrl[AxiseNo.AxisName.LCurlingneedleLine].Status.Homed AND arrAxisCtrl[AxiseNo.AxisName.LCurlingneedleLine].Status.NoMoving THEN
											IF arrAxisCtrl[AxiseNo.AxisName.LCurlingneedleLine].Cmd.arrbRealPoint[1] THEN
												arrAxisCtrl[AxiseNo.AxisName.LCurlingneedleLine].Cmd.iGoSetPos:=0;
											ELSE
												arrAxisCtrl[AxiseNo.AxisName.LCurlingneedleLine].Cmd.iGoSetPos:=1;
											END_IF
										END_IF
										IF 	arrAxisCtrl[AxiseNo.AxisName.SCurlingneedleLine].Status.Homed AND arrAxisCtrl[AxiseNo.AxisName.SCurlingneedleLine].Status.NoMoving THEN
											IF arrAxisCtrl[AxiseNo.AxisName.SCurlingneedleLine].Cmd.arrbRealPoint[1] THEN
												arrAxisCtrl[AxiseNo.AxisName.SCurlingneedleLine].Cmd.iGoSetPos:=0;
											ELSE
												arrAxisCtrl[AxiseNo.AxisName.SCurlingneedleLine].Cmd.iGoSetPos:=1;
											END_IF
										END_IF
										IF  arrAxisCtrl[AxiseNo.AxisName.LCurlingneedleLine].Cmd.arrbRealPoint[1] AND arrAxisCtrl[AxiseNo.AxisName.SCurlingneedleLine].Cmd.arrbRealPoint[1] THEN
											TON_TailCurl[3].IN:=FALSE;
											arrCyCtrl[arrCyNo.ElectValveName.WJShortvacuum].Cmd.bON:=TRUE;//短卷针张开真空开
											IF Mach_Control.WJ_b.SinStepMode THEN//尾卷单步模式
												TailCurlSinStep:=TRUE;
											ELSE
												TailCurlSinStep:=FALSE;
											END_IF												
											TailCurlStep3:=305;
										END_IF			
									END_IF
							END_IF	
							
				
							
							
							
							
							
							
							
							
							
				310://尾卷夹电芯平移至初始位
						IF NOT TailCurlSinStep THEN				
								IF 	arrCyCtrl[arrCyNo.CylinderName.TailCurlSplintCy].Io.DIOnSwitch AND  arrAxisCtrl[AxiseNo.AxisName.TailCurlLine].Status.Homed AND arrAxisCtrl[AxiseNo.AxisName.TailCurlLine].Status.NoMoving AND
                                         arrAxisCtrl[AxiseNo.AxisName.LCurlingneedleLine].Cmd.arrbRealPoint[1]  AND arrAxisCtrl[AxiseNo.AxisName.SCurlingneedleLine].Cmd.arrbRealPoint[1]  THEN
									IF arrAxisCtrl[AxiseNo.AxisName.TailCurlLine].Cmd.arrbRealPoint[1] THEN
										arrAxisCtrl[AxiseNo.AxisName.TailCurlLine].Cmd.iGoSetPos:=0;
											IF Mach_Control.WJ_b.SinStepMode THEN//尾卷单步模式
												TailCurlSinStep:=TRUE;
											ELSE
												TailCurlSinStep:=FALSE;
											END_IF										
										TailCurlStep3:=315;
									ELSE
										arrAxisCtrl[AxiseNo.AxisName.TailCurlLine].Cmd.iGoSetPos:=1;//尾卷夹电芯平移至初始位
									END_IF
								END_IF
						END_IF
				
					
						
						315://尾卷夹电芯升降至下电芯位      
						  IF NOT TailCurlSinStep THEN		                                                                                                                                                                                                                                                                                                                                                                                                   		
									IF arrAxisCtrl[AxiseNo.AxisName.TailCurlUpDown].Status.Homed AND arrAxisCtrl[AxiseNo.AxisName.TailCurlUpDown].Status.NoMoving THEN
										IF arrAxisCtrl[AxiseNo.AxisName.TailCurlUpDown].Cmd.arrbRealPoint[3] THEN
											arrAxisCtrl[AxiseNo.AxisName.TailCurlUpDown].Cmd.iGoSetPos:=0;
											IF Mach_Control.WJ_b.SinStepMode THEN//尾卷单步模式
												TailCurlSinStep:=TRUE;
											ELSE
												TailCurlSinStep:=FALSE;
											END_IF									
											TailCurlStep3:=320;
										ELSE
											arrAxisCtrl[AxiseNo.AxisName.TailCurlUpDown].Cmd.iGoSetPos:=3;//尾卷夹电芯升降至下电芯位
										END_IF
									END_IF
							END_IF	
						
						
						
						
				320://尾卷夹电芯旋转至下电芯位
						IF NOT TailCurlSinStep THEN				
								IF 	arrCyCtrl[arrCyNo.CylinderName.TailCurlSplintCy].Status.ONState AND  arrAxisCtrl[AxiseNo.AxisName.TailCurlLine].Status.Homed 
									AND arrAxisCtrl[AxiseNo.AxisName.TailCurlLine].Status.NoMoving AND arrAxisCtrl[AxiseNo.AxisName.GluingLine].Status.Homed AND
									arrAxisCtrl[AxiseNo.AxisName.GluingLine].Status.fActPos<=arrAxispar[AxiseNo.AxisName.GluingLine].arrTargetPoint[10] 
									AND NOT Mach_Control.TJ_b.StickerFlag  THEN
									IF arrAxisCtrl[AxiseNo.AxisName.TailCurlWhirling].Cmd.arrbRealPoint[2] THEN
										arrAxisCtrl[AxiseNo.AxisName.TailCurlWhirling].Cmd.iGoSetPos:=0;
											IF Mach_Control.WJ_b.SinStepMode THEN//尾卷单步模式
												TailCurlSinStep:=TRUE;
											ELSE
												TailCurlSinStep:=FALSE;
											END_IF										
										TailCurlStep3:=325;
									ELSE
										arrAxisCtrl[AxiseNo.AxisName.TailCurlWhirling].Cmd.iGoSetPos:=2;//尾卷夹电芯平移至下电芯位
									END_IF
								END_IF
						END_IF		
						
				
						
			
				325:
				//尾卷夹电芯去避让位   
					(*	  IF NOT TailCurlSinStep THEN		                                                                                                                                                                                                                                                                                                                                                                                                   		
									IF arrAxisCtrl[AxiseNo.AxisName.TailCurlLine].Status.Homed AND arrAxisCtrl[AxiseNo.AxisName.TailCurlLine].Status.NoMoving THEN
										IF arrAxisCtrl[AxiseNo.AxisName.TailCurlLine].Cmd.arrbRealPoint[5] THEN
											arrAxisCtrl[AxiseNo.AxisName.TailCurlLine].Cmd.iGoSetPos:=0;
											IF Mach_Control.WJ_b.SinStepMode THEN//尾卷单步模式
												TailCurlSinStep:=TRUE;
											ELSE
												TailCurlSinStep:=FALSE;
											END_IF									
											TailCurlStep3:=330;
										ELSE
											arrAxisCtrl[AxiseNo.AxisName.TailCurlLine].Cmd.iGoSetPos:=5;//尾卷夹电芯平移至避让位
										END_IF
									END_IF
							END_IF*)
				//尾卷夹电芯去下料避让位
							IF NOT TailCurlSinStep THEN		                                                                                                                                                                                                                                                                                                                                                                                                   		
									IF arrAxisCtrl[AxiseNo.AxisName.TailCurlLine].Status.Homed AND arrAxisCtrl[AxiseNo.AxisName.TailCurlLine].Status.NoMoving THEN
										IF arrAxisCtrl[AxiseNo.AxisName.TailCurlLine].Cmd.arrbRealPoint[10] THEN
											arrAxisCtrl[AxiseNo.AxisName.TailCurlLine].Cmd.iGoSetPos:=0;
											IF Mach_Control.WJ_b.SinStepMode THEN//尾卷单步模式
												TailCurlSinStep:=TRUE;
											ELSE
												TailCurlSinStep:=FALSE;
											END_IF									
											TailCurlStep3:=330;
										ELSE
											arrAxisCtrl[AxiseNo.AxisName.TailCurlLine].Cmd.iGoSetPos:=10;//尾卷夹电芯平移至避让位
										END_IF
									END_IF
							END_IF
				330:
						IF NOT TailCurlSinStep THEN
								Mach_Control.WJ_b.TailCultOffloading:=TRUE;//下电芯请求														
								TailCurlStep3:=332;
								
								IF Mach_Control.WJ_b.SinStepMode THEN//尾卷单步模式
									TailCurlSinStep:=TRUE;
								ELSE
									TailCurlSinStep:=FALSE;
								END_IF					
						END_IF				
						

				332:   ///////////////////
						
					IF 	arrAxisCtrl[AxiseNo.AxisName.GluingLine].Cmd.arrbRealPoint[8] AND arrAxisCtrl[AxiseNo.AxisName.GluingLine].Status.NoMoving
						AND arrAxisCtrl[AxiseNo.AxisName.GluingWhirling].Cmd.arrbRealPoint[5] AND arrAxisCtrl[AxiseNo.AxisName.GluingWhirling].Status.NoMoving
						AND arrCyCtrl[arrCyNo.CylinderName.PullGlueModelCy].Status.ONState AND NOT arrCyCtrl[arrCyNo.CylinderName.PullGlueModelCy].Status.Error2 
						AND arrAxisCtrl[AxiseNo.AxisName.TailCurlLine].Status.Homed AND arrAxisCtrl[AxiseNo.AxisName.TailCurlLine].Status.NoMoving	
						AND NOT Mach_Control.TJ_b.StickerDone  AND NOT Mach_Control.TJ_b.StickerFlag
						AND NOT CellMemory[Mach_Control.TJ_b.TJ_Memory].Cell AND NOT Mach_Control.se.GluebHave	THEN
						TailCurlStep3:=335;

					END_IF
						
				335:
						IF arrAxisCtrl[AxiseNo.AxisName.TailCurlLine].Cmd.arrbRealPoint[6] THEN
							arrAxisCtrl[AxiseNo.AxisName.TailCurlLine].Cmd.iGoSetPos:=0;
							IF Mach_Control.WJ_b.SinStepMode THEN//尾卷单步模式
								TailCurlSinStep:=TRUE;
							ELSE
								TailCurlSinStep:=FALSE;
							END_IF									
							TailCurlStep3:=336;
						ELSE
							arrAxisCtrl[AxiseNo.AxisName.TailCurlLine].Cmd.iGoSetPos:=6;//尾卷夹电芯平移至下电芯位
						END_IF
						
				336:
							IF NOT TailCurlSinStep THEN		
									IF 	arrAxisCtrl[AxiseNo.AxisName.GluingLine].Cmd.arrbRealPoint[8] AND arrAxisCtrl[AxiseNo.AxisName.GluingLine].Status.NoMoving
										AND arrAxisCtrl[AxiseNo.AxisName.GluingWhirling].Cmd.arrbRealPoint[5] AND arrAxisCtrl[AxiseNo.AxisName.GluingWhirling].Status.NoMoving
										AND arrCyCtrl[arrCyNo.CylinderName.PullGlueModelCy].Status.ONState AND NOT arrCyCtrl[arrCyNo.CylinderName.PullGlueModelCy].Status.Error2 
										AND arrAxisCtrl[AxiseNo.AxisName.TailCurlRetracting].Status.Homed AND arrAxisCtrl[AxiseNo.AxisName.TailCurlRetracting].Status.NoMoving		THEN
									IF arrAxisCtrl[AxiseNo.AxisName.TailCurlRetracting].Cmd.arrbRealPoint[3] THEN
										arrAxisCtrl[AxiseNo.AxisName.TailCurlRetracting].Cmd.iGoSetPos:=0;
										IF Mach_Control.WJ_b.SinStepMode THEN//尾卷单步模式
											TailCurlSinStep:=TRUE;
										ELSE
											TailCurlSinStep:=FALSE;
										END_IF									
										TailCurlStep3:=337;
									ELSE
										arrAxisCtrl[AxiseNo.AxisName.TailCurlRetracting].Cmd.iGoSetPos:=3;//尾卷夹电芯伸缩至下电芯位
										END_IF
									END_IF
							END_IF	
				337:
							IF NOT TailCurlSinStep THEN			
								IF 	arrAxisCtrl[AxiseNo.AxisName.TailCurlUpDown].Status.Homed AND arrAxisCtrl[AxiseNo.AxisName.TailCurlUpDown].Status.NoMoving  THEN
									IF arrAxisCtrl[AxiseNo.AxisName.TailCurlUpDown].Cmd.arrbRealPoint[4] THEN
													arrAxisCtrl[AxiseNo.AxisName.TailCurlUpDown].Cmd.iGoSetPos:=0;
													IF Mach_Control.WJ_b.SinStepMode THEN//尾卷单步模式
													TailCurlSinStep:=TRUE;
													ELSE
														TailCurlSinStep:=FALSE;
													END_IF	
													TailCurlStep3:=338;
									ELSE
													arrAxisCtrl[AxiseNo.AxisName.TailCurlUpDown].Cmd.iGoSetPos:=4;//尾卷夹电芯升降至下电芯位
									END_IF
								END_IF	
						END_IF				
						
						
						
						
						
						
				338:
				
						IF NOT TailCurlSinStep THEN				
							arrCyCtrl[arrCyNo.CylinderName.PullGlueModelCy].Cmd.bOFF:=TRUE;//贴胶治具气缸闭合
							IF arrCyCtrl[arrCyNo.CylinderName.PullGlueModelCy].Status.OFFState THEN
								IF Mach_Control.WJ_b.SinStepMode THEN//尾卷单步模式
									TailCurlSinStep:=TRUE;
								ELSE
									TailCurlSinStep:=FALSE;
								END_IF										
								TailCurlStep3:=339;
							END_IF
						END_IF


				339:
				

					IF NOT TailCurlSinStep THEN				
							arrCyCtrl[arrCyNo.CylinderName.TailCurlSplintCy].Cmd.bOFF:=TRUE;//尾卷夹爪气缸打开
							IF arrCyCtrl[arrCyNo.CylinderName.TailCurlSplintCy].Status.OFFState THEN
								arrCyCtrl[arrCyNo.ElectValveName.WJ_blow].Cmd.bOFF:=TRUE;//	夹膜电芯吹气关
								IF Mach_Control.WJ_b.SinStepMode THEN//尾卷单步模式
									TailCurlSinStep:=TRUE;
								ELSE
									TailCurlSinStep:=FALSE;
								END_IF	
								Mach_Control.TJ_b.StickerFlag:=TRUE;//置位贴胶夹爪有料标记
								TailCurlStep3:=340;
							END_IF
						END_IF

				340:
					IF NOT TailCurlSinStep THEN			
						IF 	arrAxisCtrl[AxiseNo.AxisName.TailCurlUpDown].Status.Homed AND arrAxisCtrl[AxiseNo.AxisName.TailCurlUpDown].Status.NoMoving  AND
							arrAxisCtrl[AxiseNo.AxisName.TailCurlUpDown].Cmd.arrbRealPoint[4] THEN
							arrAxisPar[AxiseNo.AxisName.TailCurlUpDown].fVelocity_of_Rel := 20   ;
							arrAxisCtrl[AxiseNo.AxisName.TailCurlUpDown].Cmd.fPosition_of_Rel :=3 ;
							arrAxisCtrl[AxiseNo.AxisName.TailCurlUpDown].Cmd.bMoveRel :=  TRUE ;
						END_IF
							IF arrAxis[AxiseNo.AxisName.TailCurlUpDown].NcToPlc.SetPos-arrAxisPar[AxiseNo.AxisName.TailCurlUpDown].arrTargetPoint[4] >=3  
							AND arrAxisCtrl[AxiseNo.AxisName.TailCurlUpDown].Status.NoMoving THEN
								IF Mach_Control.WJ_b.SinStepMode THEN//尾卷单步模式
									TailCurlSinStep:=TRUE;
								ELSE
									TailCurlSinStep:=FALSE;
								END_IF
								TailCurlStep3:=341;
							END_IF
					END_IF	
							
				341:// 尾卷夹电芯平移至避让位

						IF NOT TailCurlSinStep THEN			
								IF 	arrAxisCtrl[AxiseNo.AxisName.TailCurlLine].Status.Homed AND arrAxisCtrl[AxiseNo.AxisName.TailCurlLine].Status.NoMoving THEN
									IF arrAxisCtrl[AxiseNo.AxisName.TailCurlLine].Cmd.arrbRealPoint[10] THEN
										arrAxisCtrl[AxiseNo.AxisName.TailCurlLine].Cmd.iGoSetPos:=0;
									IF Mach_Control.WJ_b.SinStepMode THEN//尾卷单步模式
									TailCurlSinStep:=TRUE;
								ELSE
									TailCurlSinStep:=FALSE;
								END_IF	
										TailCurlStep3:=343;
									ELSE
										arrAxisCtrl[AxiseNo.AxisName.TailCurlLine].Cmd.iGoSetPos:=10;//尾卷夹电芯平移至避让位
									END_IF
								END_IF	
						END_IF	
				343:	
					CellMemory[Mach_Control.TJ_b.TJ_Memory]:=CellMemory[Mach_Control.WJ_b.WJ_Memory];
					MEMSET(ADR(CellMemory[Mach_Control.WJ_b.WJ_Memory]),0,SIZEOF(CellMemory[Mach_Control.WJ_b.WJ_Memory]));		
					TailCurlStep3:=345;		
						
						
						
						
						
						
						
				345:
		
						IF NOT TailCurlSinStep THEN			
								IF 	arrAxisCtrl[AxiseNo.AxisName.TailCurlRetracting].Status.Homed AND arrAxisCtrl[AxiseNo.AxisName.TailCurlRetracting].Status.NoMoving THEN
									IF arrAxisCtrl[AxiseNo.AxisName.TailCurlRetracting].Cmd.arrbRealPoint[1] THEN
										arrAxisCtrl[AxiseNo.AxisName.TailCurlRetracting].Cmd.iGoSetPos:=0;
										IF Mach_Control.WJ_b.SinStepMode THEN//尾卷单步模式
									TailCurlSinStep:=TRUE;
								ELSE
									TailCurlSinStep:=FALSE;
								END_IF	
										
										TailCurlStep3:=350;
									ELSE
										arrAxisCtrl[AxiseNo.AxisName.TailCurlRetracting].Cmd.iGoSetPos:=1;//尾卷夹电芯伸缩回到初始位
									END_IF
								END_IF	
						END_IF	
						
						
						
						
				350:
				IF NOT TailCurlSinStep THEN		
					 IF arrAxisCtrl[AxiseNo.AxisName.GluingLine].Status.fActPos<=arrAxispar[AxiseNo.AxisName.GluingLine].arrTargetPoint[10] 
						AND arrAxisCtrl[AxiseNo.AxisName.GluingLine].Status.Homed AND NOT Mach_Control.WJ_b.TailCultOffloading AND arrAxisCtrl[AxiseNo.AxisName.TailCurlLine].Status.Homed 
						AND arrAxisCtrl[AxiseNo.AxisName.TailCurlLine].Status.NoMoving THEN
						
								IF arrAxisCtrl[AxiseNo.AxisName.TailCurlLine].Cmd.arrbRealPoint[1] THEN
									IF Mach_Control.WJ_b.SinStepMode THEN//尾卷单步模式
									TailCurlSinStep:=TRUE;
								ELSE
									TailCurlSinStep:=FALSE;
								END_IF	
									arrAxisCtrl[AxiseNo.AxisName.TailCurlLine].Cmd.iGoSetPos:=0;
									
									TailCurlStep3:=355;
								ELSE
									arrAxisCtrl[AxiseNo.AxisName.TailCurlLine].Cmd.iGoSetPos:=1;//尾卷夹电芯平移至初始位
								END_IF
						END_IF	
				END_IF	

				355:
							IF NOT TailCurlSinStep THEN			
								IF 	arrAxisCtrl[AxiseNo.AxisName.TailCurlUpDown].Status.Homed AND arrAxisCtrl[AxiseNo.AxisName.TailCurlUpDown].Status.NoMoving  THEN
									IF arrAxisCtrl[AxiseNo.AxisName.TailCurlUpDown].Cmd.arrbRealPoint[4] THEN
													arrAxisCtrl[AxiseNo.AxisName.TailCurlUpDown].Cmd.iGoSetPos:=0;
													IF Mach_Control.WJ_b.SinStepMode THEN//尾卷单步模式
													TailCurlSinStep:=TRUE;
													ELSE
														TailCurlSinStep:=FALSE;
													END_IF	
													TailCurlStep3:=360;
									ELSE
													arrAxisCtrl[AxiseNo.AxisName.TailCurlUpDown].Cmd.iGoSetPos:=4;//尾卷夹电芯升降至下电芯位
									END_IF
								END_IF	
						END_IF
				360:
					IF NOT TailCurlSinStep THEN		
					 IF arrAxisCtrl[AxiseNo.AxisName.GluingLine].Status.fActPos<=arrAxispar[AxiseNo.AxisName.GluingLine].arrTargetPoint[10] 
						AND arrAxisCtrl[AxiseNo.AxisName.GluingLine].Status.Homed AND NOT Mach_Control.WJ_b.TailCultOffloading AND arrAxis[AxiseNo.AxisName.TailCurlWhirling].Status.Homed 
						AND arrAxisCtrl[AxiseNo.AxisName.TailCurlWhirling].Status.NoMoving AND arrAxisCtrl[AxiseNo.AxisName.TailCurlLine].Status.NoMoving AND arrAxisCtrl[AxiseNo.AxisName.TailCurlLine].Cmd.arrbRealPoint[1] THEN
						
								IF arrAxisCtrl[AxiseNo.AxisName.TailCurlWhirling].Cmd.arrbRealPoint[1] THEN
									IF Mach_Control.WJ_b.SinStepMode THEN//尾卷单步模式
									TailCurlSinStep:=TRUE;
								ELSE
									TailCurlSinStep:=FALSE;
								END_IF	
									arrAxisCtrl[AxiseNo.AxisName.TailCurlWhirling].Cmd.iGoSetPos:=0;
									//Mach_Control.WJ_b.TailCultOffloadingDone:=TRUE;
									TailCurlStep3:=370;
								ELSE
									arrAxisCtrl[AxiseNo.AxisName.TailCurlWhirling].Cmd.iGoSetPos:=1;//尾卷夹电芯旋转至取电芯位
								END_IF
						END_IF	
				END_IF	
                
				 370://尾卷夹电芯平移去取电芯等待位
					 IF NOT TailCurlSinStep THEN	
							 IF  arrAxisCtrl[AxiseNo.AxisName.TailCurlUpDown].Status.Homed AND arrAxisCtrl[AxiseNo.AxisName.TailCurlUpDown].Status.NoMoving THEN
											IF arrAxisCtrl[AxiseNo.AxisName.TailCurlUpDown].Cmd.arrbRealPoint[1] THEN
												arrAxisCtrl[AxiseNo.AxisName.TailCurlUpDown].Cmd.iGoSetPos:=0;
											ELSE
												arrAxisCtrl[AxiseNo.AxisName.TailCurlUpDown].Cmd.iGoSetPos:=1;//尾卷夹升降去取电芯高度
											END_IF
							 END_IF
						 
						   IF arrAxisCtrl[AxiseNo.AxisName.TailCurlWhirling].Cmd.arrbRealPoint[1] AND arrAxisCtrl[AxiseNo.AxisName.TailCurlUpDown].Cmd.arrbRealPoint[1] AND
							  arrAxisCtrl[AxiseNo.AxisName.TailCurlSEPTALine].Cmd.arrbRealPoint[1] AND  arrAxisCtrl[AxiseNo.AxisName.TailCurlSEPTAUpDown].Cmd.arrbRealPoint[1] AND
							  arrAxisCtrl[AxiseNo.AxisName.LCurlingneedleLine].Cmd.arrbRealPoint[1] AND arrAxisCtrl[AxiseNo.AxisName.SCurlingneedleLine].Cmd.arrbRealPoint[1] AND
							  arrCyCtrl[arrCyNo.CylinderName.PoleSplintCy_D].Io.DIOFFSwitch AND arrCyCtrl[arrCyNo.CylinderName.TailCurlUpdownCy].Io.DIOFFSwitch AND
							  arrAxisCtrl[AxiseNo.AxisName.TailCurlLine].Status.Homed AND arrAxisCtrl[AxiseNo.AxisName.TailCurlLine].Status.NoMoving  THEN
								   IF arrAxisCtrl[AxiseNo.AxisName.TailCurlLine].Cmd.arrbRealPoint[11]  THEN
									  arrAxisCtrl[AxiseNo.AxisName.TailCurlLine].Cmd.iGoSetPos:=0;
										IF Mach_Control.WJ_b.SinStepMode THEN//尾卷单步模式
										   TailCurlSinStep:=TRUE;
										ELSE
										   TailCurlSinStep:=FALSE;
										END_IF									
										   TailCurlStep3:=0;
										   TailCurlTorMark:=FALSE;//尾卷夹电芯平移力矩判断标志位
								   ELSE
									   arrAxisCtrl[AxiseNo.AxisName.TailCurlLine].Cmd.iGoSetPos:=11;//尾卷夹电芯平移去取电芯等待位
									   TailCurlTorMark:=TRUE;//尾卷夹电芯平移力矩判断标志位
								   END_IF   
							END_IF
						END_IF
				//////////////////////////////////////////////////////////////////////////////////////
				///////////////////////////////////叠台空叠隔膜不尾卷/////////////////////////////////////////////////////
				900:
					    IF NOT TailCurlSinStep THEN
							IF  Mach_Control.DT_b.OffloadRequest AND DP_Step0=6040  THEN
								IF 	arrAxisCtrl[AxiseNo.AxisName.TailCurlUpDown].Status.Homed AND arrAxisCtrl[AxiseNo.AxisName.TailCurlUpDown].Status.NoMoving THEN
										IF arrAxisCtrl[AxiseNo.AxisName.TailCurlUpDown].Cmd.arrbRealPoint[1] THEN//尾卷夹电芯升降初始位
											arrAxisCtrl[AxiseNo.AxisName.TailCurlUpDown].Cmd.iGoSetPos:=0;
										ELSE
											arrAxisCtrl[AxiseNo.AxisName.TailCurlUpDown].Cmd.iGoSetPos:=1;
										END_IF
									END_IF	
								IF 	arrAxisCtrl[AxiseNo.AxisName.TailCurlSEPTAUpDown].Status.Homed AND arrAxisCtrl[AxiseNo.AxisName.TailCurlSEPTAUpDown].Status.NoMoving THEN
										IF arrAxisCtrl[AxiseNo.AxisName.TailCurlSEPTAUpDown].Cmd.arrbRealPoint[1] THEN//夹膜升降初始位
											arrAxisCtrl[AxiseNo.AxisName.TailCurlSEPTAUpDown].Cmd.iGoSetPos:=0;
										ELSE
											arrAxisCtrl[AxiseNo.AxisName.TailCurlSEPTAUpDown].Cmd.iGoSetPos:=1;
										END_IF
									END_IF	
									IF 	arrAxisCtrl[AxiseNo.AxisName.TailCurlUpDown].Cmd.arrbRealPoint[1]  AND arrAxisCtrl[AxiseNo.AxisName.TailCurlUpDown].Cmd.arrbRealPoint[1] 
										AND arrAxisCtrl[AxiseNo.AxisName.TailCurlSEPTAUpDown].Cmd.arrbRealPoint[1]  AND arrAxisCtrl[AxiseNo.AxisName.TailCurlSEPTAUpDown].Cmd.arrbRealPoint[1]	THEN
										IF Mach_Control.WJ_b.SinStepMode THEN//尾卷单步模式
											TailCurlSinStep:=TRUE;
										ELSE
											TailCurlSinStep:=FALSE;
										END_IF								
										TailCurlStep3:=1010;	
										TON_TailCurl[6].IN:=FALSE;
									END_IF
							ELSE
								TailCurlStep3:=0;
							END_IF	
					END_IF
					
				
				
				
				/////////////////////////////////////////////////////////////////////////////////////////////////////
				/////////////////////////////////////////////////////////////////////////////////////////////////////////
				(*1000:
					Par.stDT_date.BH_Thickness :=((Par.stDT_date.An_Thickness+Par.stDT_date.SEPTA_Thickness)*Par.stDT_date.An_Quantity+(Par.stDT_date.Ca_Thickness+Par.stDT_date.SEPTA_Thickness)*Par.stDT_date.Ca_Quantity)-((Par.stDT_date.An_Thickness+Par.stDT_date.SEPTA_Thickness)*Mach_Control.An_b.An_Quantited+(Par.stDT_date.Ca_Thickness+Par.stDT_date.SEPTA_Thickness)*Mach_Control.Ca_b.Ca_Quantited);
					TailCurlStep3:=1001;

				1001:
					arrAxispar[AxiseNo.AxisName.TailCurlUpDown].arrTargetPoint[6]:=arrAxispar[AxiseNo.AxisName.TailCurlUpDown].arrTargetPoint[1]-Par.stDT_date.BH_Thickness;
					arrAxispar[AxiseNo.AxisName.TailCurlSEPTAUpDown].arrTargetPoint[3]:=arrAxispar[AxiseNo.AxisName.TailCurlSEPTAUpDown].arrTargetPoint[1]+Par.stDT_date.BH_Thickness;
					TailCurlStep3:=1005;*)




				1000://夹膜升降去取电芯位，夹电芯升降去取电芯位	
						
					    IF NOT TailCurlSinStep THEN
							IF  Mach_Control.DT_b.OffloadRequest THEN
								IF 	arrAxisCtrl[AxiseNo.AxisName.TailCurlUpDown].Status.Homed AND arrAxisCtrl[AxiseNo.AxisName.TailCurlUpDown].Status.NoMoving THEN
										IF arrAxisCtrl[AxiseNo.AxisName.TailCurlUpDown].Cmd.arrbRealPoint[6] THEN
											arrAxisCtrl[AxiseNo.AxisName.TailCurlUpDown].Cmd.iGoSetPos:=0;
										ELSE
											arrAxisCtrl[AxiseNo.AxisName.TailCurlUpDown].Cmd.iGoSetPos:=6;
										END_IF
									END_IF	
								IF 	arrAxisCtrl[AxiseNo.AxisName.TailCurlSEPTAUpDown].Status.Homed AND arrAxisCtrl[AxiseNo.AxisName.TailCurlSEPTAUpDown].Status.NoMoving THEN
										IF arrAxisCtrl[AxiseNo.AxisName.TailCurlSEPTAUpDown].Cmd.arrbRealPoint[3] THEN
											arrAxisCtrl[AxiseNo.AxisName.TailCurlSEPTAUpDown].Cmd.iGoSetPos:=0;
										ELSE
											arrAxisCtrl[AxiseNo.AxisName.TailCurlSEPTAUpDown].Cmd.iGoSetPos:=3;
										END_IF
									END_IF	
									IF 	arrAxisCtrl[AxiseNo.AxisName.TailCurlUpDown].Cmd.arrbRealPoint[6]  AND arrAxisCtrl[AxiseNo.AxisName.TailCurlUpDown].Status.NoMoving
										AND arrAxisCtrl[AxiseNo.AxisName.TailCurlSEPTAUpDown].Cmd.arrbRealPoint[3]  AND arrAxisCtrl[AxiseNo.AxisName.TailCurlSEPTAUpDown].Status.NoMoving	THEN
										IF Mach_Control.WJ_b.SinStepMode THEN//尾卷单步模式
											TailCurlSinStep:=TRUE;
										ELSE
											TailCurlSinStep:=FALSE;
										END_IF								
										TailCurlStep3:=1010;	
									END_IF
								ELSE
								TailCurlStep3:=0;
								END_IF	
					END_IF
					
		
					
				1010://负极叠片搬运平移轴在安全位置，尾卷夹电芯平移至取电芯位 、尾卷夹电芯伸缩至取电芯位 、尾卷夹膜平移至隔膜切断位///////////////////
	                 IF    NOT TailCurlSinStep AND  arrAxisCtrl[AxiseNo.AxisName.TailCurlLine].Status.Homed AND arrAxisCtrl[AxiseNo.AxisName.TailCurlLine].Status.NoMoving AND  
                           arrAxisCtrl[AxiseNo.AxisName.CaDTCarryingLine].Cmd.arrbRealPoint[1] AND arrAxisCtrl[AxiseNo.AxisName.CaDTCarryingUpDown].Cmd.arrbRealPoint[5] AND
                             arrAxisCtrl[AxiseNo.AxisName.TailCurlWhirling].Cmd.arrbRealPoint[1] AND arrAxisCtrl[AxiseNo.AxisName.SEPTATLine].Cmd.arrbRealPoint[1] AND
							 arrAxisCtrl[AxiseNo.AxisName.TailCurlSEPTAUpDown].Cmd.arrbRealPoint[3] AND arrAxisCtrl[AxiseNo.AxisName.TailCurlUpDown].Cmd.arrbRealPoint[6] AND
							  arrAxisCtrl[AxiseNo.AxisName.LCurlingneedleLine].Cmd.arrbRealPoint[1]  AND arrAxisCtrl[AxiseNo.AxisName.SCurlingneedleLine].Cmd.arrbRealPoint[1]   AND
							arrCyCtrl[arrCyNo.CylinderName.TailCurlSplintCy].Status.OFFState AND arrCyCtrl[arrCyNo.CylinderName.PoleSplintCy_D].Status.OFFState  AND
                            arrCyCtrl[arrCyNo.CylinderName.PoleHotCutterCy].Status.OFFState   THEN			
			
									IF 	 Mach_Control.DT_b.OffloadRequest THEN	
										TailCurlStep3:=1016;		
										(*	
											arrAxisCtrl[AxiseNo.AxisName.TailCurlSEPTALine].Cmd.fOverride:=100;
											arrAxisCtrl[AxiseNo.AxisName.TailCurlRetracting].Cmd.fOverride:=100;
											arrAxisCtrl[AxiseNo.AxisName.TailCurlLine].Cmd.fOverride:=100;
											
											IF   arrAxis[AxiseNo.AxisName.TailCurlSEPTALine].Status.Homed AND arrAxisCtrl[AxiseNo.AxisName.TailCurlSEPTALine].Status.NoMoving THEN
												IF arrAxisCtrl[AxiseNo.AxisName.TailCurlSEPTALine].Cmd.arrbRealPoint[2] THEN
													arrAxisCtrl[AxiseNo.AxisName.TailCurlSEPTALine].Cmd.iGoSetPos:=0;
												ELSE
													arrAxisCtrl[AxiseNo.AxisName.TailCurlSEPTALine].Cmd.iGoSetPos:=2;//尾卷夹隔膜平移取芯位
												END_IF
											END_IF
											IF 	arrAxisCtrl[AxiseNo.AxisName.TailCurlRetracting].Status.Homed AND arrAxisCtrl[AxiseNo.AxisName.TailCurlRetracting].Status.NoMoving THEN
												IF arrAxisCtrl[AxiseNo.AxisName.TailCurlRetracting].Cmd.arrbRealPoint[2] THEN
													arrAxisCtrl[AxiseNo.AxisName.TailCurlRetracting].Cmd.iGoSetPos:=0;
												ELSE
													arrAxisCtrl[AxiseNo.AxisName.TailCurlRetracting].Cmd.iGoSetPos:=2;//尾卷夹电芯伸缩至取电芯位
												END_IF
											END_IF					
											IF 	arrAxisCtrl[AxiseNo.AxisName.TailCurlLine].Status.Homed AND arrAxisCtrl[AxiseNo.AxisName.TailCurlLine].Status.NoMoving THEN
												IF arrAxisCtrl[AxiseNo.AxisName.TailCurlLine].Cmd.arrbRealPoint[2] THEN
													arrAxisCtrl[AxiseNo.AxisName.TailCurlLine].Cmd.iGoSetPos:=0;
												ELSE
													arrAxisCtrl[AxiseNo.AxisName.TailCurlLine].Cmd.iGoSetPos:=2;//尾卷夹电芯平移至取电芯位
												END_IF
											END_IF						
											IF arrAxisCtrl[AxiseNo.AxisName.TailCurlSEPTALine].Cmd.arrbRealPoint[2] AND arrAxisCtrl[AxiseNo.AxisName.TailCurlRetracting].Cmd.arrbRealPoint[2] AND
												arrAxisCtrl[AxiseNo.AxisName.TailCurlLine].Cmd.arrbRealPoint[2]  THEN
												IF  Mach_Control.WJ_b.SinStepMode THEN//尾卷单步模式
													TailCurlSinStep:=TRUE;
												ELSE
													TailCurlSinStep:=FALSE;
												END_IF	
												TailCurlStep3:=1020;
												TailCurlSplintCy_TON.IN:=FALSE;	
											END_IF
										*)
									ELSE
										TailCurlStep3:=0;
									END_IF	
						ELSE
										Mach_Control.WJ_b.Error[11]:=TRUE;	//尾卷夹电芯平移至取电芯位时条件不满足报警									
						END_IF	

				1016:
					tailCurlGearInEnable1:=TRUE;//夹电芯平移与夹膜平移电子齿轮----取料
					tailRetGearInEnable:=TRUE;//夹电芯平移与夹电芯伸缩电子齿轮
					IF tailCurl_GearIn1.InGear AND tailRetGearIn.InGear THEN
						TailCurlStep3:=1017;
					END_IF			
				1017:
					IF 	arrAxisCtrl[AxiseNo.AxisName.TailCurlLine].Status.Homed AND 
                           arrAxisCtrl[AxiseNo.AxisName.CaDTCarryingLine].Cmd.arrbRealPoint[1] AND arrAxisCtrl[AxiseNo.AxisName.CaDTCarryingUpDown].Cmd.arrbRealPoint[5] AND
                             arrAxisCtrl[AxiseNo.AxisName.TailCurlWhirling].Cmd.arrbRealPoint[1] AND arrAxisCtrl[AxiseNo.AxisName.SEPTATLine].Cmd.arrbRealPoint[1] AND
							 arrAxisCtrl[AxiseNo.AxisName.TailCurlSEPTAUpDown].Cmd.arrbRealPoint[3] AND arrAxisCtrl[AxiseNo.AxisName.TailCurlUpDown].Cmd.arrbRealPoint[6] AND
							  arrAxisCtrl[AxiseNo.AxisName.LCurlingneedleLine].Cmd.arrbRealPoint[1]  AND arrAxisCtrl[AxiseNo.AxisName.SCurlingneedleLine].Cmd.arrbRealPoint[1]   AND
							arrCyCtrl[arrCyNo.CylinderName.TailCurlSplintCy].Status.OFFState AND arrCyCtrl[arrCyNo.CylinderName.PoleSplintCy_D].Status.OFFState  AND
                            arrCyCtrl[arrCyNo.CylinderName.PoleHotCutterCy].Status.OFFState       THEN
									IF arrAxisCtrl[AxiseNo.AxisName.TailCurlLine].Cmd.arrbRealPoint[2] AND arrAxisCtrl[AxiseNo.AxisName.TailCurlLine].Status.NoMoving THEN
										TailCurlTorMark:=FALSE;//尾卷夹电芯平移力矩判断标志位
										arrAxisCtrl[AxiseNo.AxisName.TailCurlLine].Cmd.iGoSetPos:=0;
										TailCurlStep3:=1018;
									ELSE
										arrAxisCtrl[AxiseNo.AxisName.TailCurlLine].Cmd.iGoSetPos:=2;//尾卷夹电芯平移至取电芯位
										TailCurlTorMark:=TRUE;//尾卷夹电芯平移力矩判断标志位
									END_IF
					ELSE
										Mach_Control.WJ_b.Error[11]:=TRUE;	//尾卷夹电芯平移至取电芯位时条件不满足报警
					END_IF		
				1018:
					IF arrAxisCtrl[AxiseNo.AxisName.TailCurlSEPTALine].Cmd.arrbRealPoint[2] AND arrAxisCtrl[AxiseNo.AxisName.TailCurlRetracting].Cmd.arrbRealPoint[2] AND
						arrAxisCtrl[AxiseNo.AxisName.TailCurlLine].Cmd.arrbRealPoint[2]  THEN
						tailCurlGearInEnable1:=FALSE;//夹电芯平移与夹膜平移电子齿轮----取料
						tailRetGearInEnable:=FALSE;//夹电芯平移与夹电芯伸缩电子齿轮
					END_IF
					IF NOT tailCurl_GearIn1.InGear AND NOT tailRetGearIn.InGear THEN
						TailCurlStep3:=1020;
					END_IF			




				
				1020://尾卷夹电芯气缸夹紧//////////////////////////////
						arrAxisCtrl[AxiseNo.AxisName.TailCurlSEPTALine].Cmd.fOverride:=100;
						arrAxisCtrl[AxiseNo.AxisName.TailCurlRetracting].Cmd.fOverride:=100;
						arrAxisCtrl[AxiseNo.AxisName.TailCurlLine].Cmd.fOverride:=100;
						IF NOT TailCurlSinStep THEN					
							arrCyCtrl[arrCyNo.CylinderName.TailCurlSplintCy].Cmd.bON:=TRUE;//尾卷取料夹爪气缸夹紧
							TailCurlSplintCy_TON.IN:=TRUE;					
							IF (*arrCyCtrl[arrCyNo.CylinderName.TailCurlSplintCy].Io.DIOnSwitch OR*) TailCurlSplintCy_TON.Q THEN
								IF Mach_Control.WJ_b.SinStepMode THEN//尾卷单步模式
									TailCurlSinStep:=TRUE;
								ELSE
									TailCurlSinStep:=FALSE;
								END_IF								
								TailCurlStep3:=1030;
								Mach_Control.DT_b.OffloadRequest:=FALSE;//复位电芯下料请求
								TailCurlSplintCy_TON.IN:=FALSE;	
							END_IF
						END_IF
				1030://叠台升降下降至下电芯位	
					IF NOT TailCurlSinStep THEN				
								IF 	arrAxisCtrl[AxiseNo.AxisName.DTUpDown].Status.Homed   THEN
										arrAxisCtrl[AxiseNo.AxisName.DTUpDown].Cmd.bHome:=FALSE;//叠台升降下降至下电芯位回原点
												IF arrAxisCtrl[AxiseNo.AxisName.DTUpDown].Status.NoMoving THEN
															IF arrAxisCtrl[AxiseNo.AxisName.DTUpDown].Cmd.arrbRealPoint[2] THEN
																arrAxisCtrl[AxiseNo.AxisName.DTUpDown].Cmd.iGoSetPos:=0;
																IF Mach_Control.WJ_b.SinStepMode THEN//尾卷单步模式
																	TailCurlSinStep:=TRUE;
																ELSE
																	TailCurlSinStep:=FALSE;
																END_IF									
																TailCurlStep3:=1040;
															ELSE
																arrAxisCtrl[AxiseNo.AxisName.DTUpDown].Cmd.iGoSetPos:=2;//叠台升降下降至下电芯位
															END_IF
											END_IF
								ELSE
										arrAxisCtrl[AxiseNo.AxisName.DTUpDown].Cmd.bHome:=TRUE;//叠台升降下降至下电芯位回原点
								END_IF	
					END_IF
				1040://左、右压刀升降轴上升至抽刀高度
						IF NOT TailCurlSinStep THEN						
								IF 	arrAxisCtrl[AxiseNo.AxisName.LeftYDUpDown].Status.Homed AND arrAxisCtrl[AxiseNo.AxisName.LeftYDUpDown].Status.NoMoving THEN
									IF arrAxisCtrl[AxiseNo.AxisName.LeftYDUpDown].Cmd.arrbRealPoint[4] THEN
										arrAxisCtrl[AxiseNo.AxisName.LeftYDUpDown].Cmd.iGoSetPos:=0;
									ELSE
										arrAxisCtrl[AxiseNo.AxisName.LeftYDUpDown].Cmd.iGoSetPos:=4;//左压刀升降轴上升至抽刀高度
									END_IF
								END_IF					
								IF 	arrAxisCtrl[AxiseNo.AxisName.RightYDUpDown].Status.Homed AND arrAxisCtrl[AxiseNo.AxisName.RightYDUpDown].Status.NoMoving THEN
									IF arrAxisCtrl[AxiseNo.AxisName.RightYDUpDown].Cmd.arrbRealPoint[4] THEN
										arrAxisCtrl[AxiseNo.AxisName.RightYDUpDown].Cmd.iGoSetPos:=0;
									ELSE
										arrAxisCtrl[AxiseNo.AxisName.RightYDUpDown].Cmd.iGoSetPos:=4;//右压好升降上升至抽刀高度
									END_IF
								END_IF				
								IF arrAxisCtrl[AxiseNo.AxisName.LeftYDUpDown].Cmd.arrbRealPoint[4] AND arrAxisCtrl[AxiseNo.AxisName.RightYDUpDown].Cmd.arrbRealPoint[4] THEN
									IF Mach_Control.WJ_b.SinStepMode THEN//尾卷单步模式
										TailCurlSinStep:=TRUE;
									ELSE
										TailCurlSinStep:=FALSE;
									END_IF	
									TailCurlStep3:=1050;
								END_IF
						END_IF
				1050://左、右压刀开合轴至张开位
						IF NOT TailCurlSinStep THEN					
								IF 	arrAxisCtrl[AxiseNo.AxisName.LeftYDLine].Status.Homed AND arrAxisCtrl[AxiseNo.AxisName.LeftYDLine].Status.NoMoving THEN
									IF arrAxisCtrl[AxiseNo.AxisName.LeftYDLine].Cmd.arrbRealPoint[2] THEN
										arrAxisCtrl[AxiseNo.AxisName.LeftYDLine].Cmd.iGoSetPos:=0;
									ELSE
										arrAxisCtrl[AxiseNo.AxisName.LeftYDLine].Cmd.iGoSetPos:=2;//左压刀开合至张开位
									END_IF
								END_IF					
								IF 	arrAxisCtrl[AxiseNo.AxisName.RightYDLine].Status.Homed AND arrAxisCtrl[AxiseNo.AxisName.RightYDLine].Status.NoMoving THEN
									IF arrAxisCtrl[AxiseNo.AxisName.RightYDLine].Cmd.arrbRealPoint[3] THEN
										arrAxisCtrl[AxiseNo.AxisName.RightYDLine].Cmd.iGoSetPos:=0;
									ELSE
										arrAxisCtrl[AxiseNo.AxisName.RightYDLine].Cmd.iGoSetPos:=3;//右压刀开合至张开位
									END_IF
								END_IF				
								IF arrAxisCtrl[AxiseNo.AxisName.LeftYDLine].Cmd.arrbRealPoint[2] AND arrAxisCtrl[AxiseNo.AxisName.RightYDLine].Cmd.arrbRealPoint[3] THEN
									IF Mach_Control.WJ_b.SinStepMode THEN//尾卷单步模式
										TailCurlSinStep:=TRUE;
									ELSE
										TailCurlSinStep:=FALSE;
									END_IF										
									TailCurlStep3:=1060;
								END_IF	
						END_IF
						
				1060:
						IF NOT TailCurlSinStep THEN		
								IF 	arrAxisCtrl[AxiseNo.AxisName.RightYDUpDown].Status.Homed AND arrAxisCtrl[AxiseNo.AxisName.RightYDUpDown].Status.NoMoving THEN
									IF arrAxisCtrl[AxiseNo.AxisName.RightYDUpDown].Cmd.arrbRealPoint[5] THEN
										arrAxisCtrl[AxiseNo.AxisName.RightYDUpDown].Cmd.iGoSetPos:=0;
									ELSE
										arrAxisCtrl[AxiseNo.AxisName.RightYDUpDown].Cmd.iGoSetPos:=5;//右压好升降上升至下料张开位
									END_IF
								END_IF				
								IF  arrAxisCtrl[AxiseNo.AxisName.RightYDUpDown].Cmd.arrbRealPoint[5] THEN
									IF Mach_Control.WJ_b.SinStepMode THEN//尾卷单步模式
										TailCurlSinStep:=TRUE;
									ELSE
										TailCurlSinStep:=FALSE;
									END_IF	
									TailCurlStep3:=1070;
								END_IF

						END_IF
		
				1065:
					
						(*IF NOT TailCurlSinStep THEN	
							arrCyCtrl[arrCyNo.CylinderName.PreDiaph].Cmd.bON:=TRUE;//叠台压隔膜气缸
							IF arrCyCtrl[arrCyNo.CylinderName.PreDiaph].Status.ONState THEN
								IF Mach_Control.WJ_b.SinStepMode THEN//尾卷单步模式
									TailCurlSinStep:=TRUE;
								ELSE
									TailCurlSinStep:=FALSE;
								END_IF									
								TailCurlStep3:=1070;	
							END_IF	
						END_IF	*)			
									
						
				1070://尾卷夹电芯平移至拉膜位、尾卷夹电芯伸缩至初始位、
						IF NOT TailCurlSinStep THEN	
							tailCult_GearInMultiMaster.Enable:=TRUE;//启动尾卷拉膜凸轮耦合
							fbGearInGMvirbEnable:=TRUE;//尾卷拉膜纠偏
							arrAxisCtrl[AxiseNo.AxisName.TailCurlLine].Cmd.fOverride:=30;
							arrAxisCtrl[AxiseNo.AxisName.TailCurlRetracting].Cmd.fOverride:=30;
							IF  tailCult_GearInMultiMaster.InGear THEN
								
							
										IF 	arrAxisCtrl[AxiseNo.AxisName.TailCurlRetracting].Status.Homed AND arrAxisCtrl[AxiseNo.AxisName.TailCurlRetracting].Status.NoMoving THEN
										
											IF arrAxisCtrl[AxiseNo.AxisName.TailCurlRetracting].Cmd.arrbRealPoint[1] THEN
												arrAxisCtrl[AxiseNo.AxisName.TailCurlRetracting].Cmd.iGoSetPos:=0;
											ELSE
												arrAxisCtrl[AxiseNo.AxisName.TailCurlRetracting].Cmd.iGoSetPos:=1;//尾卷夹电芯伸缩移至初始位
											END_IF
										END_IF				
									
										IF 	arrAxisCtrl[AxiseNo.AxisName.TailCurlLine].Status.Homed AND arrAxisCtrl[AxiseNo.AxisName.TailCurlLine].Status.NoMoving AND
                                               arrAxisCtrl[AxiseNo.AxisName.LCurlingneedleLine].Cmd.arrbRealPoint[1]  AND arrAxisCtrl[AxiseNo.AxisName.SCurlingneedleLine].Cmd.arrbRealPoint[1]  THEN
											IF arrAxisCtrl[AxiseNo.AxisName.TailCurlLine].Cmd.arrbRealPoint[9] THEN
												arrAxisCtrl[AxiseNo.AxisName.TailCurlLine].Cmd.iGoSetPos:=0;
											ELSE
												arrAxisCtrl[AxiseNo.AxisName.TailCurlLine].Cmd.iGoSetPos:=9;//尾卷夹电芯平移至对齐度NG切膜位
											END_IF
										END_IF																		
									IF 	arrAxisCtrl[AxiseNo.AxisName.TailCurlRetracting].Cmd.arrbRealPoint[1] AND arrAxisCtrl[AxiseNo.AxisName.TailCurlLine].Cmd.arrbRealPoint[9]  THEN
											tailCult_GearInMultiMaster.Enable:=FALSE;//启动尾卷拉膜凸轮耦合
											IF Mach_Control.WJ_b.SinStepMode THEN//尾卷单步模式
												TailCurlSinStep:=TRUE;
											ELSE
												TailCurlSinStep:=FALSE;
											END_IF
											fbGearInGMvirbEnable	:=FALSE;
											arrAxisCtrl[AxiseNo.AxisName.TailCurlLine].Cmd.fOverride:=100;
											arrAxisCtrl[AxiseNo.AxisName.TailCurlRetracting].Cmd.fOverride:=100;									
											TailCurlStep3:=1075;
											NGcount:=NGcount+1;
								END_IF	
						END_IF
						END_IF
		

					1075:	
							arrAxisCtrl[AxiseNo.AxisName.TailCurlLine].Cmd.fOverride:=100;
							arrAxisCtrl[AxiseNo.AxisName.TailCurlRetracting].Cmd.fOverride:=100;
							IF NOT TailCurlSinStep THEN			
										IF arrAxis[AxiseNo.AxisName.TailCurlWhirling].Status.Homed AND arrAxisCtrl[AxiseNo.AxisName.TailCurlWhirling].Status.NoMoving THEN
													IF arrAxisCtrl[AxiseNo.AxisName.TailCurlWhirling].Cmd.arrbRealPoint[4] THEN
														arrAxisCtrl[AxiseNo.AxisName.TailCurlWhirling].Cmd.iGoSetPos:=0;
														IF Mach_Control.WJ_b.SinStepMode THEN//尾卷单步模式
															TailCurlSinStep:=TRUE;
														ELSE
															TailCurlSinStep:=FALSE;
														END_IF	
														TailCurlStep3:=1080;
													ELSE
														arrAxisCtrl[AxiseNo.AxisName.TailCurlWhirling].Cmd.iGoSetPos:=4;
													END_IF						
									END_IF
								END_IF
						
	
						
					1080://左、右压刀开合至张开位
						IF NOT TailCurlSinStep THEN		
								
								IF 	arrAxisCtrl[AxiseNo.AxisName.LeftYDUpDown].Status.Homed AND arrAxisCtrl[AxiseNo.AxisName.LeftYDUpDown].Status.NoMoving THEN
									IF arrAxisCtrl[AxiseNo.AxisName.LeftYDUpDown].Cmd.arrbRealPoint[2] THEN
										arrAxisCtrl[AxiseNo.AxisName.LeftYDUpDown].Cmd.iGoSetPos:=0;
									ELSE
										arrAxisCtrl[AxiseNo.AxisName.LeftYDUpDown].Cmd.iGoSetPos:=2;//左压刀升降轴上升至下料高度
									END_IF
								END_IF					
								IF 	arrAxisCtrl[AxiseNo.AxisName.RightYDUpDown].Status.Homed AND arrAxisCtrl[AxiseNo.AxisName.RightYDUpDown].Status.NoMoving THEN
									IF arrAxisCtrl[AxiseNo.AxisName.RightYDUpDown].Cmd.arrbRealPoint[2] THEN
										arrAxisCtrl[AxiseNo.AxisName.RightYDUpDown].Cmd.iGoSetPos:=0;
									ELSE
										arrAxisCtrl[AxiseNo.AxisName.RightYDUpDown].Cmd.iGoSetPos:=2;//右压好升降上升至下料高度
									END_IF
								END_IF																	
								IF 	arrAxisCtrl[AxiseNo.AxisName.TailCurlSEPTAUpDown].Status.Homed AND arrAxisCtrl[AxiseNo.AxisName.TailCurlSEPTAUpDown].Status.NoMoving THEN
									IF arrAxisCtrl[AxiseNo.AxisName.TailCurlSEPTAUpDown].Cmd.arrbRealPoint[2] THEN
										arrAxisCtrl[AxiseNo.AxisName.TailCurlSEPTAUpDown].Cmd.iGoSetPos:=0;
									ELSE
										arrAxisCtrl[AxiseNo.AxisName.TailCurlSEPTAUpDown].Cmd.iGoSetPos:=2;//
									END_IF
								END_IF					
								IF 	arrAxisCtrl[AxiseNo.AxisName.TailCurlUpDown].Status.Homed AND arrAxisCtrl[AxiseNo.AxisName.TailCurlUpDown].Status.NoMoving THEN
									IF arrAxisCtrl[AxiseNo.AxisName.TailCurlUpDown].Cmd.arrbRealPoint[2] THEN
										arrAxisCtrl[AxiseNo.AxisName.TailCurlUpDown].Cmd.iGoSetPos:=0;
									ELSE
										arrAxisCtrl[AxiseNo.AxisName.TailCurlUpDown].Cmd.iGoSetPos:=2;//
									END_IF
								END_IF									
								
								IF  arrAxisCtrl[AxiseNo.AxisName.TailCurlUpDown].Cmd.arrbRealPoint[2] AND arrAxisCtrl[AxiseNo.AxisName.TailCurlSEPTAUpDown].Cmd.arrbRealPoint[2] AND
									arrAxisCtrl[AxiseNo.AxisName.LeftYDUpDown].Cmd.arrbRealPoint[2] AND arrAxisCtrl[AxiseNo.AxisName.RightYDUpDown].Cmd.arrbRealPoint[2]  THEN
									IF Mach_Control.WJ_b.SinStepMode THEN//尾卷单步模式
										TailCurlSinStep:=TRUE;
									ELSE
										TailCurlSinStep:=FALSE;
									END_IF		
									TailCurlStep3:=1085;
								END_IF
						END_IF		
				1085:
						IF NOT TailCurlSinStep THEN	
							arrCyCtrl[arrCyNo.ElectValveName.PoleSplintVacuum_D].Cmd.bON:=TRUE;//夹膜下夹板真空	
							arrCyCtrl[arrCyNo.CylinderName.PoleSplintCy_D].Cmd.bON:=TRUE;//夹膜下夹板上升
								IF arrCyCtrl[arrCyNo.CylinderName.PoleSplintCy_D].Status.ONState THEN
									IF Mach_Control.WJ_b.SinStepMode THEN//尾卷单步模式
										TailCurlSinStep:=TRUE;
									ELSE
										TailCurlSinStep:=FALSE;
									END_IF									
									TailCurlStep3:=1090;	
								END_IF	
						END_IF	
	
				1090:
					
						IF NOT TailCurlSinStep THEN	
							arrCyCtrl[arrCyNo.CylinderName.PreDiaph].Cmd.bON:=TRUE;//叠台压隔膜气缸
							IF arrCyCtrl[arrCyNo.CylinderName.PreDiaph].Status.ONState THEN
								IF Mach_Control.WJ_b.SinStepMode THEN//尾卷单步模式
									TailCurlSinStep:=TRUE;
								ELSE
									TailCurlSinStep:=FALSE;
								END_IF									
								TailCurlStep3:=1100;
							END_IF	
						END_IF							
			


				1100://左、右压刀开合移至初始位，叠台上升至初始位
						IF NOT TailCurlSinStep THEN		
									IF 	arrAxisCtrl[AxiseNo.AxisName.LeftYDLine].Status.Homed AND arrAxisCtrl[AxiseNo.AxisName.LeftYDLine].Status.NoMoving THEN
										IF arrAxisCtrl[AxiseNo.AxisName.LeftYDLine].Cmd.arrbRealPoint[1] THEN
											arrAxisCtrl[AxiseNo.AxisName.LeftYDLine].Cmd.iGoSetPos:=0;
										ELSE
											arrAxisCtrl[AxiseNo.AxisName.LeftYDLine].Cmd.iGoSetPos:=1;//左压刀开合至初始位
										END_IF
									END_IF					
									IF 	arrAxisCtrl[AxiseNo.AxisName.RightYDLine].Status.Homed AND arrAxisCtrl[AxiseNo.AxisName.RightYDLine].Status.NoMoving THEN
										IF arrAxisCtrl[AxiseNo.AxisName.RightYDLine].Cmd.arrbRealPoint[1] THEN
											arrAxisCtrl[AxiseNo.AxisName.RightYDLine].Cmd.iGoSetPos:=0;
										ELSE
											arrAxisCtrl[AxiseNo.AxisName.RightYDLine].Cmd.iGoSetPos:=1;//右压刀开合至初始位
										END_IF
									END_IF
									IF 	arrAxisCtrl[AxiseNo.AxisName.DTUpDown].Status.Homed AND arrAxisCtrl[AxiseNo.AxisName.DTUpDown].Status.NoMoving THEN
										IF arrAxisCtrl[AxiseNo.AxisName.DTUpDown].Cmd.arrbRealPoint[1] THEN
											arrAxisCtrl[AxiseNo.AxisName.DTUpDown].Cmd.iGoSetPos:=0;
										ELSE
											arrAxisCtrl[AxiseNo.AxisName.DTUpDown].Cmd.iGoSetPos:=1;//叠台升降上升至初始位
										END_IF
									END_IF
									IF 	arrAxisCtrl[AxiseNo.AxisName.LeftYDLine].Cmd.arrbRealPoint[1] AND arrAxisCtrl[AxiseNo.AxisName.RightYDLine].Cmd.arrbRealPoint[1] AND 
										arrAxisCtrl[AxiseNo.AxisName.DTUpDown].Cmd.arrbRealPoint[1] THEN
												TailCurlStep3:=1110;
												IF Mach_Control.WJ_b.SinStepMode THEN//尾卷单步模式
													TailCurlSinStep:=TRUE;
												ELSE
													TailCurlSinStep:=FALSE;
												END_IF	
									END_IF	
						END_IF
				
					



				1110://左、右压刀升降下降至初始位，压隔膜
						IF NOT TailCurlSinStep THEN			
									IF 	arrAxisCtrl[AxiseNo.AxisName.LeftYDUpDown].Status.Homed AND arrAxisCtrl[AxiseNo.AxisName.LeftYDUpDown].Status.NoMoving THEN
										IF arrAxisCtrl[AxiseNo.AxisName.LeftYDUpDown].Cmd.arrbRealPoint[1] THEN
											arrAxisCtrl[AxiseNo.AxisName.LeftYDUpDown].Cmd.iGoSetPos:=0;
										ELSE
											arrAxisCtrl[AxiseNo.AxisName.LeftYDUpDown].Cmd.iGoSetPos:=1;//左压刀升降轴下降至初始高度
										END_IF
									END_IF					
									IF 	arrAxisCtrl[AxiseNo.AxisName.RightYDUpDown].Status.Homed AND arrAxisCtrl[AxiseNo.AxisName.RightYDUpDown].Status.NoMoving THEN
										IF arrAxisCtrl[AxiseNo.AxisName.RightYDUpDown].Cmd.arrbRealPoint[1] THEN
											arrAxisCtrl[AxiseNo.AxisName.RightYDUpDown].Cmd.iGoSetPos:=0;
										ELSE
											arrAxisCtrl[AxiseNo.AxisName.RightYDUpDown].Cmd.iGoSetPos:=1;//右压好升降下降至初始高度
										END_IF
									END_IF				
									IF arrAxisCtrl[AxiseNo.AxisName.LeftYDUpDown].Cmd.arrbRealPoint[1] AND arrAxisCtrl[AxiseNo.AxisName.RightYDUpDown].Cmd.arrbRealPoint[1] THEN
										IF Mach_Control.WJ_b.SinStepMode THEN//尾卷单步模式
											TailCurlSinStep:=TRUE;
										ELSE
											TailCurlSinStep:=FALSE;
										END_IF											
										TailCurlStep3:=1120;
										hot_time_ton.IN:=FALSE;
									END_IF
						END_IF
						
					(*1120:
						Mach_Control.WJ_b.HotCut:=TRUE;//启动热切
						WJ_TON[1].IN:=TRUE;
						TailCurlStep3:=1130;		
					
						
				1130://热切丝加热、热切升降气缸下降，切隔膜///////////////////////////////
					IF NOT TailCurlSinStep THEN	
					arrCyCtrl[arrCyNo.CylinderName.PoleHotCutterCy].Cmd.bON:=TRUE;//隔膜热切升降气缸伸出
								IF arrCyCtrl[arrCyNo.CylinderName.PoleHotCutterCy].Status.ONState  THEN
										Mach_Control.WJ_b.HotCut:=FALSE;//启动热切
						                WJ_TON[1].IN:=FALSE;
							IF Mach_Control.WJ_b.SinStepMode THEN//尾卷单步模式
								TailCurlSinStep:=TRUE;
							ELSE
								TailCurlSinStep:=FALSE;
							END_IF							
									TailCurlStep3:=1140;	
								END_IF	
					END_IF*)	
				
				1140://热切升降气缸下降/////////////////////////////////////////
				IF NOT TailCurlSinStep THEN	
					Blueflaging:=FALSE;
					arrCyCtrl[arrCyNo.CylinderName.PoleHotCutterCy].Cmd.bOFF:=TRUE;//隔膜热切升降气缸缩回	
						IF arrCyCtrl[arrCyNo.CylinderName.PoleHotCutterCy].Status.OFFState THEN
							IF Mach_Control.WJ_b.SinStepMode THEN//尾卷单步模式
								TailCurlSinStep:=TRUE;
							ELSE
								TailCurlSinStep:=FALSE;
							END_IF									
							TailCurlStep3:=1142;	
						END_IF	
				END_IF	

				1142://叠台真空打开
					arrCyCtrl[arrCyNo.ElectValveName.DTVacuum].Cmd.bON:=TRUE;
					arrCyCtrl[arrCyNo.ElectValveName.DTVacuum].Cmd.bOFF:=FALSE;
					TailCurlStep3:=1145;
					
				1145:
						IF NOT TailCurlSinStep THEN	
							arrCyCtrl[arrCyNo.ElectValveName.PoleSplintVacuum_D].Cmd.bOFF:=TRUE;//夹膜下夹板真空	
							arrCyCtrl[arrCyNo.CylinderName.PoleSplintCy_D].Cmd.bOFF:=TRUE;//夹膜下夹板上升
								IF arrCyCtrl[arrCyNo.CylinderName.PoleSplintCy_D].Status.OFFState THEN
									IF Mach_Control.WJ_b.SinStepMode THEN//尾卷单步模式
										TailCurlSinStep:=TRUE;
									ELSE
										TailCurlSinStep:=FALSE;
									END_IF									
									TailCurlStep3:=1148;	
								END_IF	
						END_IF							
				
				1148:
					IF 	arrAxisCtrl[AxiseNo.AxisName.TailCurlSEPTAUpDown].Status.Homed AND arrAxisCtrl[AxiseNo.AxisName.TailCurlSEPTAUpDown].Status.NoMoving THEN
						IF arrAxisCtrl[AxiseNo.AxisName.TailCurlSEPTAUpDown].Cmd.arrbRealPoint[1] THEN
							arrAxisCtrl[AxiseNo.AxisName.TailCurlSEPTAUpDown].Cmd.iGoSetPos:=0;
						ELSE
							arrAxisCtrl[AxiseNo.AxisName.TailCurlSEPTAUpDown].Cmd.iGoSetPos:=1;//
						END_IF
					END_IF
					IF arrAxisCtrl[AxiseNo.AxisName.TailCurlSEPTAUpDown].Cmd.arrbRealPoint[1] THEN
						TailCurlStep3:=1150;	
					END_IF
	

				1150:
					CellMemory[Mach_Control.WJ_b.WJ_Memory]:=CellMemory[Mach_Control.DT_b.DT_Memory];
					MEMSET(ADR(CellMemory[Mach_Control.DT_b.DT_Memory]),0,SIZEOF(CellMemory[Mach_Control.DT_b.DT_Memory]));
					TailCurlStep3:=1160;
		
				1160:
					
						IF NOT TailCurlSinStep THEN	
							arrCyCtrl[arrCyNo.CylinderName.PreDiaph].Cmd.bOFF:=TRUE;//
							IF arrCyCtrl[arrCyNo.CylinderName.PreDiaph].Status.OFFState THEN
								IF Mach_Control.WJ_b.SinStepMode THEN//尾卷单步模式
									TailCurlSinStep:=TRUE;
								ELSE
									TailCurlSinStep:=FALSE;
								END_IF									
								TailCurlStep3:=1170;
								TailCurlStep6:=10;//启动判断夹膜平移是否已经在安全位置叠台下料完成	
							END_IF	
						END_IF

				1170:
					IF NOT TailCurlSinStep THEN	
					
						IF 	arrAxisCtrl[AxiseNo.AxisName.TailCurlLine].Status.Homed AND arrAxisCtrl[AxiseNo.AxisName.TailCurlLine].Status.NoMoving AND
                                arrAxisCtrl[AxiseNo.AxisName.LCurlingneedleLine].Cmd.arrbRealPoint[1]  AND arrAxisCtrl[AxiseNo.AxisName.SCurlingneedleLine].Cmd.arrbRealPoint[1] AND
                                 arrAxisCtrl[AxiseNo.AxisName.TailCurlWhirling].Cmd.arrbRealPoint[1]  THEN
								IF arrAxisCtrl[AxiseNo.AxisName.TailCurlLine].Cmd.arrbRealPoint[1] THEN
									arrAxisCtrl[AxiseNo.AxisName.TailCurlLine].Cmd.iGoSetPos:=0;
								ELSE
									arrAxisCtrl[AxiseNo.AxisName.TailCurlLine].Cmd.iGoSetPos:=1;//尾卷夹电芯平移至初始位
								END_IF
							END_IF	
						IF   arrAxis[AxiseNo.AxisName.TailCurlSEPTALine].Status.Homed AND arrAxisCtrl[AxiseNo.AxisName.TailCurlSEPTALine].Status.NoMoving AND arrAxisCtrl[AxiseNo.AxisName.TailCurlLine].Status.Homed 
								AND arrAxisCtrl[AxiseNo.AxisName.TailCurlLine].Status.fActPos<arrAxisPar[AxiseNo.AxisName.TailCurlLine].arrTargetPoint[7] THEN
								IF arrAxisCtrl[AxiseNo.AxisName.TailCurlSEPTALine].Cmd.arrbRealPoint[1] THEN
									arrAxisCtrl[AxiseNo.AxisName.TailCurlSEPTALine].Cmd.iGoSetPos:=0;
								ELSE
									arrAxisCtrl[AxiseNo.AxisName.TailCurlSEPTALine].Cmd.iGoSetPos:=1;//尾卷夹隔膜平移至初始位
								END_IF
						END_IF
						IF arrAxisCtrl[AxiseNo.AxisName.TailCurlLine].Cmd.arrbRealPoint[1] AND arrAxisCtrl[AxiseNo.AxisName.TailCurlLine].Status.NoMoving 
							AND arrAxisCtrl[AxiseNo.AxisName.TailCurlSEPTALine].Cmd.arrbRealPoint[1] AND  arrAxisCtrl[AxiseNo.AxisName.TailCurlSEPTALine].Status.NoMoving AND
							TailCurlStep6=666  THEN
								IF Mach_Control.WJ_b.SinStepMode THEN//尾卷单步模式
									TailCurlSinStep:=TRUE;
								ELSE
									TailCurlSinStep:=FALSE;
								END_IF									
								TailCurlStep3:=1180;
							END_IF
					END_IF
				1180://尾卷夹电芯升降至下电芯位      
						  IF NOT TailCurlSinStep THEN		                                                                                                                                                                                                                                                                                                                                                                                                   		
									IF arrAxisCtrl[AxiseNo.AxisName.TailCurlUpDown].Status.Homed AND arrAxisCtrl[AxiseNo.AxisName.TailCurlUpDown].Status.NoMoving THEN
										IF arrAxisCtrl[AxiseNo.AxisName.TailCurlUpDown].Cmd.arrbRealPoint[3] THEN
											arrAxisCtrl[AxiseNo.AxisName.TailCurlUpDown].Cmd.iGoSetPos:=0;	
										ELSE
											arrAxisCtrl[AxiseNo.AxisName.TailCurlUpDown].Cmd.iGoSetPos:=3;//尾卷夹电芯升降至下电芯位
										END_IF
									END_IF
							IF 	arrAxisCtrl[AxiseNo.AxisName.TailCurlSEPTAUpDown].Status.Homed AND arrAxisCtrl[AxiseNo.AxisName.TailCurlSEPTAUpDown].Status.NoMoving THEN
								IF arrAxisCtrl[AxiseNo.AxisName.TailCurlSEPTAUpDown].Cmd.arrbRealPoint[1] THEN
									arrAxisCtrl[AxiseNo.AxisName.TailCurlSEPTAUpDown].Cmd.iGoSetPos:=0;
								ELSE
									arrAxisCtrl[AxiseNo.AxisName.TailCurlSEPTAUpDown].Cmd.iGoSetPos:=1;
								END_IF
							END_IF
							IF arrAxisCtrl[AxiseNo.AxisName.TailCurlUpDown].Cmd.arrbRealPoint[3] AND arrAxisCtrl[AxiseNo.AxisName.TailCurlUpDown].Status.NoMoving
								AND arrAxisCtrl[AxiseNo.AxisName.TailCurlSEPTAUpDown].Cmd.arrbRealPoint[1] AND  arrAxisCtrl[AxiseNo.AxisName.TailCurlSEPTAUpDown].Status.NoMoving THEN
								IF Mach_Control.WJ_b.SinStepMode THEN//尾卷单步模式
												TailCurlSinStep:=TRUE;
											ELSE
												TailCurlSinStep:=FALSE;
											END_IF									
											TailCurlStep3:=1190;
							END_IF	
						END_IF
						
						
						
				1190://尾卷夹电芯旋转至下电芯位
						IF NOT TailCurlSinStep THEN				
								IF 	(*arrCyCtrl[arrCyNo.CylinderName.TailCurlSplintCy].Status.ONState AND*)  arrAxisCtrl[AxiseNo.AxisName.TailCurlLine].Status.Homed 
									AND arrAxisCtrl[AxiseNo.AxisName.TailCurlLine].Status.NoMoving AND arrAxisCtrl[AxiseNo.AxisName.GluingLine].Status.Homed AND
									arrAxisCtrl[AxiseNo.AxisName.GluingLine].Status.fActPos<=arrAxispar[AxiseNo.AxisName.GluingLine].arrTargetPoint[10] 
									AND NOT Mach_Control.TJ_b.StickerFlag  THEN
									IF arrAxisCtrl[AxiseNo.AxisName.TailCurlWhirling].Cmd.arrbRealPoint[2] THEN
										arrAxisCtrl[AxiseNo.AxisName.TailCurlWhirling].Cmd.iGoSetPos:=0;
											IF Mach_Control.WJ_b.SinStepMode THEN//尾卷单步模式
												TailCurlSinStep:=TRUE;
											ELSE
												TailCurlSinStep:=FALSE;
											END_IF										
										TailCurlStep3:=1200;
									ELSE
										arrAxisCtrl[AxiseNo.AxisName.TailCurlWhirling].Cmd.iGoSetPos:=2;//尾卷夹电芯平移至下电芯位
									END_IF
								END_IF
						END_IF		
						
				
						
			
				1200:
				//尾卷夹电芯去下料避让位   
						  IF NOT TailCurlSinStep THEN		                                                                                                                                                                                                                                                                                                                                                                                                   		
									IF arrAxisCtrl[AxiseNo.AxisName.TailCurlLine].Status.Homed AND arrAxisCtrl[AxiseNo.AxisName.TailCurlLine].Status.NoMoving THEN
										IF arrAxisCtrl[AxiseNo.AxisName.TailCurlLine].Cmd.arrbRealPoint[10] THEN
											arrAxisCtrl[AxiseNo.AxisName.TailCurlLine].Cmd.iGoSetPos:=0;
											IF Mach_Control.WJ_b.SinStepMode THEN//尾卷单步模式
												TailCurlSinStep:=TRUE;
											ELSE
												TailCurlSinStep:=FALSE;
											END_IF									
											TailCurlStep3:=1210;
										ELSE
											arrAxisCtrl[AxiseNo.AxisName.TailCurlLine].Cmd.iGoSetPos:=10;//尾卷夹电芯平移至避让位
										END_IF
									END_IF
							END_IF
				1210:
						IF NOT TailCurlSinStep THEN
								Mach_Control.WJ_b.TailCultOffloading:=TRUE;//下电芯请求														
								TailCurlStep3:=1220;
								
								IF Mach_Control.WJ_b.SinStepMode THEN//尾卷单步模式
									TailCurlSinStep:=TRUE;
								ELSE
									TailCurlSinStep:=FALSE;
								END_IF					
						END_IF				
						

				1220:   ///////////////////
						
					IF 	arrAxisCtrl[AxiseNo.AxisName.GluingLine].Cmd.arrbRealPoint[8] AND arrAxisCtrl[AxiseNo.AxisName.GluingLine].Status.NoMoving
						AND arrAxisCtrl[AxiseNo.AxisName.GluingWhirling].Cmd.arrbRealPoint[5] AND arrAxisCtrl[AxiseNo.AxisName.GluingWhirling].Status.NoMoving
						AND arrCyCtrl[arrCyNo.CylinderName.PullGlueModelCy].Status.ONState AND NOT arrCyCtrl[arrCyNo.CylinderName.PullGlueModelCy].Status.Error2 
						AND arrAxisCtrl[AxiseNo.AxisName.TailCurlLine].Status.Homed AND arrAxisCtrl[AxiseNo.AxisName.TailCurlLine].Status.NoMoving	
						AND NOT Mach_Control.TJ_b.StickerDone  AND NOT Mach_Control.TJ_b.StickerFlag
						AND NOT CellMemory[Mach_Control.TJ_b.TJ_Memory].Cell AND NOT Mach_Control.se.GluebHave	THEN
						TailCurlStep3:=1225;
					ELSIF Mach_Control.se.GluebHave AND arrAxisCtrl[AxiseNo.AxisName.GluingWhirling].Status.NoMoving THEN
						Mach_Control.TJ_b.Error[9]:=TRUE; //贴胶夹爪有信号无记忆报警
					END_IF
						
				1225:
						IF arrAxisCtrl[AxiseNo.AxisName.TailCurlLine].Cmd.arrbRealPoint[6] THEN
							arrAxisCtrl[AxiseNo.AxisName.TailCurlLine].Cmd.iGoSetPos:=0;
							IF Mach_Control.WJ_b.SinStepMode THEN//尾卷单步模式
								TailCurlSinStep:=TRUE;
							ELSE
								TailCurlSinStep:=FALSE;
							END_IF									
							TailCurlStep3:=1230;
						ELSE
							arrAxisCtrl[AxiseNo.AxisName.TailCurlLine].Cmd.iGoSetPos:=6;//尾卷夹电芯平移至下电芯位
						END_IF
						
						
				1230:
							IF NOT TailCurlSinStep THEN		
									IF 	arrAxisCtrl[AxiseNo.AxisName.GluingLine].Cmd.arrbRealPoint[8] AND arrAxisCtrl[AxiseNo.AxisName.GluingLine].Status.NoMoving
										AND arrAxisCtrl[AxiseNo.AxisName.GluingWhirling].Cmd.arrbRealPoint[5] AND arrAxisCtrl[AxiseNo.AxisName.GluingWhirling].Status.NoMoving
										AND arrCyCtrl[arrCyNo.CylinderName.PullGlueModelCy].Status.ONState AND NOT arrCyCtrl[arrCyNo.CylinderName.PullGlueModelCy].Status.Error2 
										AND arrAxisCtrl[AxiseNo.AxisName.TailCurlRetracting].Status.Homed AND arrAxisCtrl[AxiseNo.AxisName.TailCurlRetracting].Status.NoMoving		THEN
									IF arrAxisCtrl[AxiseNo.AxisName.TailCurlRetracting].Cmd.arrbRealPoint[3] THEN
										arrAxisCtrl[AxiseNo.AxisName.TailCurlRetracting].Cmd.iGoSetPos:=0;
										IF Mach_Control.WJ_b.SinStepMode THEN//尾卷单步模式
											TailCurlSinStep:=TRUE;
										ELSE
											TailCurlSinStep:=FALSE;
										END_IF									
										TailCurlStep3:=1240;
									ELSE
										arrAxisCtrl[AxiseNo.AxisName.TailCurlRetracting].Cmd.iGoSetPos:=3;//尾卷夹电芯伸缩至下电芯位
										END_IF
									END_IF
							END_IF	
				1240:
							IF NOT TailCurlSinStep THEN			
								IF 	arrAxisCtrl[AxiseNo.AxisName.TailCurlUpDown].Status.Homed AND arrAxisCtrl[AxiseNo.AxisName.TailCurlUpDown].Status.NoMoving  THEN
									IF arrAxisCtrl[AxiseNo.AxisName.TailCurlUpDown].Cmd.arrbRealPoint[4] THEN
													arrAxisCtrl[AxiseNo.AxisName.TailCurlUpDown].Cmd.iGoSetPos:=0;
													IF Mach_Control.WJ_b.SinStepMode THEN//尾卷单步模式
													TailCurlSinStep:=TRUE;
													ELSE
														TailCurlSinStep:=FALSE;
													END_IF	
													TailCurlStep3:=1260;
									ELSE
													arrAxisCtrl[AxiseNo.AxisName.TailCurlUpDown].Cmd.iGoSetPos:=4;//尾卷夹电芯升降至下电芯位
									END_IF
								END_IF	
						END_IF									
(*						
				1250:
				
						IF NOT TailCurlSinStep THEN				
							arrCyCtrl[arrCyNo.CylinderName.PullGlueModelCy].Cmd.bOFF:=TRUE;//贴胶治具气缸闭合
							IF arrCyCtrl[arrCyNo.CylinderName.PullGlueModelCy].Status.OFFState THEN
								IF Mach_Control.WJ_b.SinStepMode THEN//尾卷单步模式
									TailCurlSinStep:=TRUE;
								ELSE
									TailCurlSinStep:=FALSE;
								END_IF										
								TailCurlStep3:=1260;
							END_IF
						END_IF
*)

				1260:
				

					IF NOT TailCurlSinStep THEN				
							arrCyCtrl[arrCyNo.CylinderName.TailCurlSplintCy].Cmd.bOFF:=TRUE;//尾卷夹爪气缸打开
							IF arrCyCtrl[arrCyNo.CylinderName.TailCurlSplintCy].Status.OFFState THEN
								IF Mach_Control.WJ_b.SinStepMode THEN//尾卷单步模式
									TailCurlSinStep:=TRUE;
								ELSE
									TailCurlSinStep:=FALSE;
								END_IF	
								Mach_Control.TJ_b.StickerFlag:=TRUE;//置位贴胶夹爪有料标记
								TailCurlStep3:=1265;
							END_IF
						END_IF

				1265:
					IF NOT TailCurlSinStep THEN			
						IF 	arrAxisCtrl[AxiseNo.AxisName.TailCurlUpDown].Status.Homed AND arrAxisCtrl[AxiseNo.AxisName.TailCurlUpDown].Status.NoMoving  AND
							arrAxisCtrl[AxiseNo.AxisName.TailCurlUpDown].Cmd.arrbRealPoint[4] THEN
							arrAxisPar[AxiseNo.AxisName.TailCurlUpDown].fVelocity_of_Rel := 20   ;
							arrAxisCtrl[AxiseNo.AxisName.TailCurlUpDown].Cmd.fPosition_of_Rel :=3 ;
							arrAxisCtrl[AxiseNo.AxisName.TailCurlUpDown].Cmd.bMoveRel :=  TRUE ;
						END_IF
							IF arrAxis[AxiseNo.AxisName.TailCurlUpDown].NcToPlc.SetPos-arrAxisPar[AxiseNo.AxisName.TailCurlUpDown].arrTargetPoint[4] >=3  
							AND arrAxisCtrl[AxiseNo.AxisName.TailCurlUpDown].Status.NoMoving THEN
								IF Mach_Control.WJ_b.SinStepMode THEN//尾卷单步模式
									TailCurlSinStep:=TRUE;
								ELSE
									TailCurlSinStep:=FALSE;
								END_IF
								TailCurlStep3:=1270;
							END_IF
					END_IF	
									
							
				1270:// 尾卷夹电芯平移至下料避让位
						IF NOT TailCurlSinStep THEN			
								IF 	arrAxisCtrl[AxiseNo.AxisName.TailCurlLine].Status.Homed AND arrAxisCtrl[AxiseNo.AxisName.TailCurlLine].Status.NoMoving THEN
									IF arrAxisCtrl[AxiseNo.AxisName.TailCurlLine].Cmd.arrbRealPoint[10] THEN
										arrAxisCtrl[AxiseNo.AxisName.TailCurlLine].Cmd.iGoSetPos:=0;
									IF Mach_Control.WJ_b.SinStepMode THEN//尾卷单步模式
									TailCurlSinStep:=TRUE;
								ELSE
									TailCurlSinStep:=FALSE;
								END_IF	
										TailCurlStep3:=1280;
									ELSE
										arrAxisCtrl[AxiseNo.AxisName.TailCurlLine].Cmd.iGoSetPos:=10;//尾卷夹电芯平移至下料避让位
									END_IF
								END_IF	
						END_IF	



				1280:	
					CellMemory[Mach_Control.TJ_b.TJ_Memory]:=CellMemory[Mach_Control.WJ_b.WJ_Memory];
					MEMSET(ADR(CellMemory[Mach_Control.WJ_b.WJ_Memory]),0,SIZEOF(CellMemory[Mach_Control.WJ_b.WJ_Memory]));		
					TailCurlStep3:=1290;		
						
						
						
						
						
						
						
				1290:
		
						IF NOT TailCurlSinStep THEN			
								IF 	arrAxisCtrl[AxiseNo.AxisName.TailCurlRetracting].Status.Homed AND arrAxisCtrl[AxiseNo.AxisName.TailCurlRetracting].Status.NoMoving THEN
									IF arrAxisCtrl[AxiseNo.AxisName.TailCurlRetracting].Cmd.arrbRealPoint[1] THEN
										arrAxisCtrl[AxiseNo.AxisName.TailCurlRetracting].Cmd.iGoSetPos:=0;
										IF Mach_Control.WJ_b.SinStepMode THEN//尾卷单步模式
									TailCurlSinStep:=TRUE;
								ELSE
									TailCurlSinStep:=FALSE;
								END_IF	
										
										TailCurlStep3:=1300;
									ELSE
										arrAxisCtrl[AxiseNo.AxisName.TailCurlRetracting].Cmd.iGoSetPos:=1;//尾卷夹电芯伸缩回到初始位
									END_IF
								END_IF	
						END_IF	
						
						
						
						
				1300:
				IF NOT TailCurlSinStep THEN		
					 IF arrAxisCtrl[AxiseNo.AxisName.GluingLine].Status.fActPos<=arrAxispar[AxiseNo.AxisName.GluingLine].arrTargetPoint[10] 
						AND arrAxisCtrl[AxiseNo.AxisName.GluingLine].Status.Homed AND NOT Mach_Control.WJ_b.TailCultOffloading AND arrAxisCtrl[AxiseNo.AxisName.TailCurlLine].Status.Homed 
						AND arrAxisCtrl[AxiseNo.AxisName.TailCurlLine].Status.NoMoving THEN
						
